LIN {X 0,Y 245.646,Z 172.876,A -85,B 0,C 180,E1 -19098.135,E2 -19098.135} C_VEL
LIN {X 0,Y 243.166,Z 173.176,A -85,B 0,C 180,E1 -19099.924,E2 -19099.924} C_VEL
LIN {X 0,Y 242.08,Z 173.312,A -85,B 0,C 180,E1 -19101.313,E2 -19101.313} C_VEL
LIN {X 0,Y 241.982,Z 173.328,A -85,B 0,C 180,E1 -19101.785,E2 -19101.785} C_VEL
LIN {X 0,Y 241.988,Z 173.343,A -85,B 0,C 180,E1 -19105.826,E2 -19105.826} C_VEL
LIN {X 0,Y 241.964,Z 173.344,A -85,B 0,C 180,E1 -19109.589,E2 -19109.589} C_VEL
LIN {X 0,Y 241.98,Z 173.342,A -85,B 0,C 180,E1 -19113.493,E2 -19113.493} C_VEL
LIN {X 0,Y 241.985,Z 173.344,A -85,B 0,C 180,E1 -19117.583,E2 -19117.583} C_VEL
LIN {X 0,Y 241.909,Z 173.35,A -85,B 0,C 180,E1 -19121.928,E2 -19121.928} C_VEL
LIN {X 0,Y 241.902,Z 173.348,A -85,B 0,C 180,E1 -19126.58,E2 -19126.58} C_VEL
LIN {X 0,Y 241.993,Z 173.342,A -85,B 0,C 180,E1 -19131.641,E2 -19131.641} C_VEL
LIN {X 0,Y 242.055,Z 173.351,A -85,B 0,C 180,E1 -19133.453,E2 -19133.453} C_VEL
LIN {X 0,Y 244.108,Z 182.855,A -85,B 0,C 180,E1 -19137.329,E2 -19137.329} C_VEL
LIN {X 0,Y 244.835,Z 186.515,A -85,B 0,C 180,E1 -19138.763,E2 -19138.763} C_VEL
LIN {X 0,Y 252.464,Z 207.324,A -85,B 0,C 180,E1 -19140.307,E2 -19140.307} C_VEL
LIN {X 0,Y 256.373,Z 235.384,A -85,B 0,C 180,E1 -19141.627,E2 -19141.627} C_VEL
LIN {X 0,Y 254.176,Z 295.63,A -85,B 0,C 180,E1 -19143.433,E2 -19143.433} C_VEL
LIN {X 0,Y 253.102,Z 309.545,A -85,B 0,C 180,E1 -19144.176,E2 -19144.176} C_VEL
LIN {X 0,Y 251.698,Z 321.703,A -85,B 0,C 180,E1 -19145.129,E2 -19145.129} C_VEL
LIN {X 0,Y 250.002,Z 333.498,A -85,B 0,C 180,E1 -19146.385,E2 -19146.385} C_VEL
LIN {X 0,Y 248.104,Z 344.903,A -85,B 0,C 180,E1 -19147.955,E2 -19147.955} C_VEL
LIN {X 0,Y 246.364,Z 355.221,A -85,B 0,C 180,E1 -19149.764,E2 -19149.764} C_VEL
LIN {X 0,Y 244.557,Z 365.313,A -85,B 0,C 180,E1 -19152.005,E2 -19152.005} C_VEL
LIN {X 0,Y 242.888,Z 374.18,A -85,B 0,C 180,E1 -19154.475,E2 -19154.475} C_VEL
LIN {X 0,Y 241.493,Z 381.221,A -85,B 0,C 180,E1 -19156.965,E2 -19156.965} C_VEL
LIN {X 0,Y 240.541,Z 387.674,A -85,B 0,C 180,E1 -19159.904,E2 -19159.904} C_VEL
LIN {X 0,Y 240.047,Z 391.882,A -85,B 0,C 180,E1 -19162.429,E2 -19162.429} C_VEL
LIN {X 0,Y 239.837,Z 395.125,A -85,B 0,C 180,E1 -19165.077,E2 -19165.077} C_VEL
LIN {X 0,Y 239.798,Z 396.531,A -85,B 0,C 180,E1 -19166.64,E2 -19166.64} C_VEL
LIN {X 0,Y 239.844,Z 397.601,A -85,B 0,C 180,E1 -19168.321,E2 -19168.321} C_VEL
LIN {X 0,Y 239.913,Z 398.261,A -85,B 0,C 180,E1 -19170,E2 -19170} C_VEL
LIN {X 0,Y 239.83,Z 398.521,A -85,B 0,C 180,E1 -19171.679,E2 -19171.679} C_VEL
LIN {X 0,Y 239.791,Z 397.941,A -85,B 0,C 180,E1 -19174.792,E2 -19174.792} C_VEL
LIN {X 0,Y 239.953,Z 396.852,A -85,B 0,C 180,E1 -19176.728,E2 -19176.728} C_VEL
LIN {X 0,Y 240.668,Z 393.726,A -85,B 0,C 180,E1 -19180.091,E2 -19180.091} C_VEL
LIN {X 0,Y 241.609,Z 390.211,A -85,B 0,C 180,E1 -19182.601,E2 -19182.601} C_VEL
LIN {X 0,Y 242.969,Z 385.623,A -85,B 0,C 180,E1 -19185.09,E2 -19185.09} C_VEL
LIN {X 0,Y 245.261,Z 378.7,A -85,B 0,C 180,E1 -19187.942,E2 -19187.942} C_VEL
LIN {X 0,Y 247.484,Z 371.049,A -85,B 0,C 180,E1 -19190.425,E2 -19190.425} C_VEL
LIN {X 0,Y 250.137,Z 362.038,A -85,B 0,C 180,E1 -19192.726,E2 -19192.726} C_VEL
LIN {X 0,Y 252.83,Z 352.498,A -85,B 0,C 180,E1 -19194.643,E2 -19194.643} C_VEL
LIN {X 0,Y 255.464,Z 341.974,A -85,B 0,C 180,E1 -19196.335,E2 -19196.335} C_VEL
LIN {X 0,Y 258.126,Z 330.254,A -85,B 0,C 180,E1 -19197.792,E2 -19197.792} C_VEL
LIN {X 0,Y 260.337,Z 317.845,A -85,B 0,C 180,E1 -19198.963,E2 -19198.963} C_VEL
LIN {X 0,Y 262.108,Z 305.644,A -85,B 0,C 180,E1 -19199.795,E2 -19199.795} C_VEL
LIN {X 0,Y 263.402,Z 292.249,A -85,B 0,C 180,E1 -19200.406,E2 -19200.406} C_VEL
LIN {X 0,Y 265.957,Z 237.913,A -85,B 0,C 180,E1 -19202.004,E2 -19202.004} C_VEL
LIN {X 0,Y 263.486,Z 220.784,A -85,B 0,C 180,E1 -19203.076,E2 -19203.076} C_VEL
LIN {X 0,Y 257.206,Z 206.553,A -85,B 0,C 180,E1 -19204.794,E2 -19204.794} C_VEL
LIN {X 0,Y 251.031,Z 194.528,A -85,B 0,C 180,E1 -19206.568,E2 -19206.568} C_VEL
LIN {X 0,Y 247.245,Z 188.246,A -85,B 0,C 180,E1 -19207.687,E2 -19207.687} C_VEL
LIN {X 0,Y 245.239,Z 184.526,A -85,B 0,C 180,E1 -19208.326,E2 -19208.326} C_VEL
LIN {X 0,Y 243.191,Z 177.489,A -85,B 0,C 180,E1 -19212.12,E2 -19212.12} C_VEL
LIN {X 0,Y 241.928,Z 173.348,A -85,B 0,C 180,E1 -19214.685,E2 -19214.685} C_VEL
LIN {X 0,Y 241.914,Z 173.349,A -85,B 0,C 180,E1 -19219.056,E2 -19219.056} C_VEL
LIN {X 0,Y 241.984,Z 173.338,A -85,B 0,C 180,E1 -19222.417,E2 -19222.417} C_VEL
LIN {X 0,Y 241.981,Z 173.333,A -85,B 0,C 180,E1 -19226.507,E2 -19226.507} C_VEL
LIN {X 0,Y 241.972,Z 173.331,A -85,B 0,C 180,E1 -19230.616,E2 -19230.616} C_VEL
LIN {X 0,Y 241.997,Z 173.33,A -85,B 0,C 180,E1 -19234.198,E2 -19234.198} C_VEL
LIN {X 0,Y 241.987,Z 173.333,A -85,B 0,C 180,E1 -19238.338,E2 -19238.338} C_VEL
LIN {X 0,Y 242.108,Z 173.317,A -85,B 0,C 180,E1 -19243.325,E2 -19243.325} C_VEL
LIN {X 0,Y 242.151,Z 173.308,A -85,B 0,C 180,E1 -19248.278,E2 -19248.278} C_VEL
LIN {X 0,Y 242.389,Z 173.289,A -85,B 0,C 180,E1 -19251.664,E2 -19251.664} C_VEL
LIN {X 0,Y 242.408,Z 173.273,A -85,B 0,C 180,E1 -19253.34,E2 -19253.34} C_VEL
LIN {X 0,Y 242.618,Z 173.25,A -85,B 0,C 180,E1 -19258.34,E2 -19258.34} C_VEL
LIN {X 0,Y 242.618,Z 173.251,A -85,B 0,C 180,E1 -19261.66,E2 -19261.66} C_VEL
LIN {X 0,Y 242.403,Z 173.284,A -85,B 0,C 180,E1 -19266.66,E2 -19266.66} C_VEL
LIN {X 0,Y 242.263,Z 173.301,A -85,B 0,C 180,E1 -19270.024,E2 -19270.024} C_VEL
LIN {X 0,Y 242.109,Z 173.323,A -85,B 0,C 180,E1 -19275.145,E2 -19275.145} C_VEL
LIN {X 0,Y 242.076,Z 173.453,A -85,B 0,C 180,E1 -19277.639,E2 -19277.639} C_VEL
LIN {X 0,Y 242.773,Z 175.92,A -85,B 0,C 180,E1 -19279.116,E2 -19279.116} C_VEL
LIN {X 0,Y 245.193,Z 179.843,A -85,B 0,C 180,E1 -19279.9,E2 -19279.9} C_VEL
LIN {X 0,Y 250.376,Z 187.916,A -85,B 0,C 180,E1 -19281.458,E2 -19281.458} C_VEL
LIN {X 0,Y 256.429,Z 198.44,A -85,B 0,C 180,E1 -19283.176,E2 -19283.176} C_VEL
LIN {X 0,Y 262.613,Z 210.801,A -85,B 0,C 180,E1 -19284.837,E2 -19284.837} C_VEL
LIN {X 0,Y 266.786,Z 220.657,A -85,B 0,C 180,E1 -19285.946,E2 -19285.946} C_VEL
LIN {X 0,Y 263.559,Z 283.684,A -85,B 0,C 180,E1 -19287.801,E2 -19287.801} C_VEL
LIN {X 0,Y 262.233,Z 296.967,A -85,B 0,C 180,E1 -19288.483,E2 -19288.483} C_VEL
LIN {X 0,Y 260.633,Z 309.3,A -85,B 0,C 180,E1 -19289.433,E2 -19289.433} C_VEL
LIN {X 0,Y 258.485,Z 321.395,A -85,B 0,C 180,E1 -19290.688,E2 -19290.688} C_VEL
LIN {X 0,Y 256.148,Z 332.007,A -85,B 0,C 180,E1 -19292.098,E2 -19292.098} C_VEL
LIN {X 0,Y 253.657,Z 342.027,A -85,B 0,C 180,E1 -19293.777,E2 -19293.777} C_VEL
LIN {X 0,Y 251.1,Z 351.324,A -85,B 0,C 180,E1 -19295.739,E2 -19295.739} C_VEL
LIN {X 0,Y 248.786,Z 358.929,A -85,B 0,C 180,E1 -19297.722,E2 -19297.722} C_VEL
LIN {X 0,Y 246.429,Z 366.325,A -85,B 0,C 180,E1 -19300.131,E2 -19300.131} C_VEL
LIN {X 0,Y 244.297,Z 372.773,A -85,B 0,C 180,E1 -19302.812,E2 -19302.812} C_VEL
LIN {X 0,Y 242.383,Z 378.302,A -85,B 0,C 180,E1 -19305.901,E2 -19305.901} C_VEL
LIN {X 0,Y 241.425,Z 381.072,A -85,B 0,C 180,E1 -19307.968,E2 -19307.968} C_VEL
LIN {X 0,Y 240.702,Z 383.099,A -85,B 0,C 180,E1 -19310.032,E2 -19310.032} C_VEL
LIN {X 0,Y 240.069,Z 384.596,A -85,B 0,C 180,E1 -19312.225,E2 -19312.225} C_VEL
LIN {X 0,Y 239.587,Z 385.494,A -85,B 0,C 180,E1 -19315.22,E2 -19315.22} C_VEL
LIN {X 0,Y 239.436,Z 385.099,A -85,B 0,C 180,E1 -19318.345,E2 -19318.345} C_VEL
LIN {X 0,Y 239.493,Z 384.301,A -85,B 0,C 180,E1 -19320.074,E2 -19320.074} C_VEL
LIN {X 0,Y 239.701,Z 382.835,A -85,B 0,C 180,E1 -19322.023,E2 -19322.023} C_VEL
LIN {X 0,Y 240.304,Z 379.465,A -85,B 0,C 180,E1 -19325.045,E2 -19325.045} C_VEL
LIN {X 0,Y 240.978,Z 375.219,A -85,B 0,C 180,E1 -19327.719,E2 -19327.719} C_VEL
LIN {X 0,Y 241.958,Z 369.369,A -85,B 0,C 180,E1 -19330.486,E2 -19330.486} C_VEL
LIN {X 0,Y 243.365,Z 361.912,A -85,B 0,C 180,E1 -19333.215,E2 -19333.215} C_VEL
LIN {X 0,Y 244.887,Z 354.288,A -85,B 0,C 180,E1 -19335.433,E2 -19335.433} C_VEL
LIN {X 0,Y 246.618,Z 344.762,A -85,B 0,C 180,E1 -19337.659,E2 -19337.659} C_VEL
LIN {X 0,Y 248.535,Z 334.204,A -85,B 0,C 180,E1 -19339.614,E2 -19339.614} C_VEL
LIN {X 0,Y 250.384,Z 322.487,A -85,B 0,C 180,E1 -19341.324,E2 -19341.324} C_VEL
LIN {X 0,Y 251.952,Z 310.311,A -85,B 0,C 180,E1 -19342.688,E2 -19342.688} C_VEL
LIN {X 0,Y 253.267,Z 297.726,A -85,B 0,C 180,E1 -19343.741,E2 -19343.741} C_VEL
LIN {X 0,Y 254.329,Z 284.519,A -85,B 0,C 180,E1 -19344.485,E2 -19344.485} C_VEL
LIN {X 0,Y 255.167,Z 264.929,A -85,B 0,C 180,E1 -19345.129,E2 -19345.129} C_VEL
LIN {X 0,Y 257.003,Z 212.02,A -85,B 0,C 180,E1 -19346.679,E2 -19346.679} C_VEL
LIN {X 0,Y 251.113,Z 195.487,A -85,B 0,C 180,E1 -19347.835,E2 -19347.835} C_VEL
LIN {X 0,Y 242.82,Z 174.317,A -85,B 0,C 180,E1 -19349.534,E2 -19349.534} C_VEL
LIN {X 0,Y 242.641,Z 173.263,A -85,B 0,C 180,E1 -19350,E2 -19350} C_VEL
LIN {X 0,Y 242.623,Z 173.262,A -85,B 0,C 180,E1 -19351.66,E2 -19351.66} C_VEL
LIN {X 0,Y 242.403,Z 173.288,A -85,B 0,C 180,E1 -19356.66,E2 -19356.66} C_VEL
LIN {X 0,Y 242.268,Z 173.306,A -85,B 0,C 180,E1 -19360.024,E2 -19360.024} C_VEL
LIN {X 0,Y 242.113,Z 173.324,A -85,B 0,C 180,E1 -19365.144,E2 -19365.144} C_VEL
LIN {X 0,Y 242.046,Z 173.333,A -85,B 0,C 180,E1 -19368.626,E2 -19368.626} C_VEL
LIN {X 0,Y 241.99,Z 173.337,A -85,B 0,C 180,E1 -19372.182,E2 -19372.182} C_VEL
LIN {X 0,Y 241.988,Z 173.336,A -85,B 0,C 180,E1 -19375.826,E2 -19375.826} C_VEL
LIN {X 0,Y 241.97,Z 173.344,A -85,B 0,C 180,E1 -19379.588,E2 -19379.588} C_VEL
LIN {X 0,Y 241.981,Z 173.326,A -85,B 0,C 180,E1 -19383.493,E2 -19383.493} C_VEL
LIN {X 0,Y 241.988,Z 173.341,A -85,B 0,C 180,E1 -19387.583,E2 -19387.583} C_VEL
LIN {X 0,Y 241.911,Z 173.346,A -85,B 0,C 180,E1 -19391.928,E2 -19391.928} C_VEL
LIN {X 0,Y 241.902,Z 173.325,A -85,B 0,C 180,E1 -19396.58,E2 -19396.58} C_VEL
LIN {X 0,Y 241.995,Z 173.339,A -85,B 0,C 180,E1 -19401.641,E2 -19401.641} C_VEL
LIN {X 0,Y 241.982,Z 173.342,A -85,B 0,C 180,E1 -19404.488,E2 -19404.488} C_VEL
LIN {X 0,Y 241.955,Z 173.337,A -85,B 0,C 180,E1 -19408.477,E2 -19408.477} C_VEL
LIN {X 0,Y 241.97,Z 173.343,A -85,B 0,C 180,E1 -19412.308,E2 -19412.308} C_VEL
LIN {X 0,Y 242.026,Z 173.33,A -85,B 0,C 180,E1 -19416.012,E2 -19416.012} C_VEL
LIN {X 0,Y 241.987,Z 173.339,A -85,B 0,C 180,E1 -19419.603,E2 -19419.603} C_VEL
LIN {X 0,Y 242.108,Z 173.322,A -85,B 0,C 180,E1 -19423.324,E2 -19423.324} C_VEL
LIN {X 0,Y 242.164,Z 173.318,A -85,B 0,C 180,E1 -19428.279,E2 -19428.279} C_VEL
LIN {X 0,Y 242.388,Z 173.289,A -85,B 0,C 180,E1 -19431.664,E2 -19431.664} C_VEL
LIN {X 0,Y 242.404,Z 173.283,A -85,B 0,C 180,E1 -19433.34,E2 -19433.34} C_VEL
LIN {X 0,Y 242.62,Z 173.265,A -85,B 0,C 180,E1 -19438.34,E2 -19438.34} C_VEL
LIN {X 0,Y 242.619,Z 173.259,A -85,B 0,C 180,E1 -19441.66,E2 -19441.66} C_VEL
LIN {X 0,Y 242.399,Z 173.263,A -85,B 0,C 180,E1 -19446.66,E2 -19446.66} C_VEL
LIN {X 0,Y 242.262,Z 173.298,A -85,B 0,C 180,E1 -19450.024,E2 -19450.024} C_VEL
LIN {X 0,Y 242.104,Z 173.326,A -85,B 0,C 180,E1 -19455.145,E2 -19455.145} C_VEL
LIN {X 0,Y 242.016,Z 173.325,A -85,B 0,C 180,E1 -19458.629,E2 -19458.629} C_VEL
LIN {X 0,Y 241.982,Z 173.328,A -85,B 0,C 180,E1 -19461.785,E2 -19461.785} C_VEL
LIN {X 0,Y 241.28,Z 173.426,A -85,B 0,C 180,E1 -19463.175,E2 -19463.175} C_VEL
LIN {X 0,Y 238.396,Z 173.79,A -85,B 0,C 180,E1 -19465.442,E2 -19465.442} C_VEL
LIN {X 0,Y 235.978,Z 174.091,A -85,B 0,C 180,E1 -19467.289,E2 -19467.289} C_VEL
LIN {X 0,Y 234.964,Z 174.212,A -85,B 0,C 180,E1 -19468.723,E2 -19468.723} C_VEL
LIN {X 0,Y 234.893,Z 174.221,A -85,B 0,C 180,E1 -19469.208,E2 -19469.208} C_VEL
LIN {X 0,Y 234.942,Z 174.22,A -85,B 0,C 180,E1 -19473.113,E2 -19473.113} C_VEL
LIN {X 0,Y 234.917,Z 174.224,A -85,B 0,C 180,E1 -19476.751,E2 -19476.751} C_VEL
LIN {X 0,Y 234.913,Z 174.225,A -85,B 0,C 180,E1 -19478.935,E2 -19478.935} C_VEL
LIN {X 0,Y 234.854,Z 174.23,A -85,B 0,C 180,E1 -19483.494,E2 -19483.494} C_VEL
LIN {X 0,Y 234.855,Z 174.226,A -85,B 0,C 180,E1 -19486.506,E2 -19486.506} C_VEL
LIN {X 0,Y 234.919,Z 174.224,A -85,B 0,C 180,E1 -19491.078,E2 -19491.078} C_VEL
LIN {X 0,Y 234.993,Z 174.243,A -85,B 0,C 180,E1 -19492.861,E2 -19492.861} C_VEL
LIN {X 0,Y 237.063,Z 183.657,A -85,B 0,C 180,E1 -19496.833,E2 -19496.833} C_VEL
LIN {X 0,Y 237.643,Z 186.548,A -85,B 0,C 180,E1 -19497.927,E2 -19497.927} C_VEL
LIN {X 0,Y 246.115,Z 209.016,A -85,B 0,C 180,E1 -19499.693,E2 -19499.693} C_VEL
LIN {X 0,Y 249.791,Z 235.832,A -85,B 0,C 180,E1 -19500.997,E2 -19500.997} C_VEL
LIN {X 0,Y 247.639,Z 294.718,A -85,B 0,C 180,E1 -19502.803,E2 -19502.803} C_VEL
LIN {X 0,Y 246.541,Z 308.656,A -85,B 0,C 180,E1 -19503.55,E2 -19503.55} C_VEL
LIN {X 0,Y 245.09,Z 321.021,A -85,B 0,C 180,E1 -19504.524,E2 -19504.524} C_VEL
LIN {X 0,Y 243.504,Z 332.149,A -85,B 0,C 180,E1 -19505.714,E2 -19505.714} C_VEL
LIN {X 0,Y 241.543,Z 343.765,A -85,B 0,C 180,E1 -19507.323,E2 -19507.323} C_VEL
LIN {X 0,Y 239.639,Z 354.257,A -85,B 0,C 180,E1 -19509.17,E2 -19509.17} C_VEL
LIN {X 0,Y 237.983,Z 362.832,A -85,B 0,C 180,E1 -19511.044,E2 -19511.044} C_VEL
LIN {X 0,Y 236.495,Z 370.734,A -85,B 0,C 180,E1 -19513.157,E2 -19513.157} C_VEL
LIN {X 0,Y 234.982,Z 378.423,A -85,B 0,C 180,E1 -19515.715,E2 -19515.715} C_VEL
LIN {X 0,Y 233.779,Z 385.517,A -85,B 0,C 180,E1 -19518.731,E2 -19518.731} C_VEL
LIN {X 0,Y 233.168,Z 390.19,A -85,B 0,C 180,E1 -19521.332,E2 -19521.332} C_VEL
LIN {X 0,Y 232.896,Z 392.644,A -85,B 0,C 180,E1 -19523.067,E2 -19523.067} C_VEL
LIN {X 0,Y 232.728,Z 395.091,A -85,B 0,C 180,E1 -19525.238,E2 -19525.238} C_VEL
LIN {X 0,Y 232.756,Z 397.333,A -85,B 0,C 180,E1 -19528.27,E2 -19528.27} C_VEL
LIN {X 0,Y 232.823,Z 398.022,A -85,B 0,C 180,E1 -19530,E2 -19530} C_VEL
LIN {X 0,Y 232.742,Z 398.31,A -85,B 0,C 180,E1 -19531.73,E2 -19531.73} C_VEL
LIN {X 0,Y 232.707,Z 397.869,A -85,B 0,C 180,E1 -19534.699,E2 -19534.699} C_VEL
LIN {X 0,Y 232.891,Z 396.752,A -85,B 0,C 180,E1 -19536.933,E2 -19536.933} C_VEL
LIN {X 0,Y 233.665,Z 393.688,A -85,B 0,C 180,E1 -19540.397,E2 -19540.397} C_VEL
LIN {X 0,Y 234.644,Z 390.234,A -85,B 0,C 180,E1 -19542.982,E2 -19542.982} C_VEL
LIN {X 0,Y 236.127,Z 385.723,A -85,B 0,C 180,E1 -19545.538,E2 -19545.538} C_VEL
LIN {X 0,Y 238.511,Z 378.933,A -85,B 0,C 180,E1 -19548.467,E2 -19548.467} C_VEL
LIN {X 0,Y 240.749,Z 371.719,A -85,B 0,C 180,E1 -19550.908,E2 -19550.908} C_VEL
LIN {X 0,Y 243.622,Z 362.498,A -85,B 0,C 180,E1 -19553.37,E2 -19553.37} C_VEL
LIN {X 0,Y 246.725,Z 352.045,A -85,B 0,C 180,E1 -19555.521,E2 -19555.521} C_VEL
LIN {X 0,Y 249.52,Z 341.464,A -85,B 0,C 180,E1 -19557.239,E2 -19557.239} C_VEL
LIN {X 0,Y 252.245,Z 329.657,A -85,B 0,C 180,E1 -19558.726,E2 -19558.726} C_VEL
LIN {X 0,Y 254.564,Z 317.191,A -85,B 0,C 180,E1 -19559.912,E2 -19559.912} C_VEL
LIN {X 0,Y 256.523,Z 304.129,A -85,B 0,C 180,E1 -19560.796,E2 -19560.796} C_VEL
LIN {X 0,Y 257.782,Z 290.61,A -85,B 0,C 180,E1 -19561.392,E2 -19561.392} C_VEL
LIN {X 0,Y 260.312,Z 238.633,A -85,B 0,C 180,E1 -19562.955,E2 -19562.955} C_VEL
LIN {X 0,Y 258.26,Z 223.958,A -85,B 0,C 180,E1 -19563.902,E2 -19563.902} C_VEL
LIN {X 0,Y 252.636,Z 210.85,A -85,B 0,C 180,E1 -19565.538,E2 -19565.538} C_VEL
LIN {X 0,Y 246.677,Z 199.127,A -85,B 0,C 180,E1 -19567.332,E2 -19567.332} C_VEL
LIN {X 0,Y 240.762,Z 188.999,A -85,B 0,C 180,E1 -19569.226,E2 -19569.226} C_VEL
LIN {X 0,Y 238.016,Z 184.471,A -85,B 0,C 180,E1 -19570.159,E2 -19570.159} C_VEL
LIN {X 0,Y 236.345,Z 179.132,A -85,B 0,C 180,E1 -19573.152,E2 -19573.152} C_VEL
LIN {X 0,Y 234.862,Z 174.229,A -85,B 0,C 180,E1 -19576.277,E2 -19576.277} C_VEL
LIN {X 0,Y 234.919,Z 174.219,A -85,B 0,C 180,E1 -19581.079,E2 -19581.079} C_VEL
LIN {X 0,Y 234.927,Z 174.221,A -85,B 0,C 180,E1 -19585.361,E2 -19585.361} C_VEL
LIN {X 0,Y 234.897,Z 174.222,A -85,B 0,C 180,E1 -19589.427,E2 -19589.427} C_VEL
LIN {X 0,Y 234.941,Z 174.213,A -85,B 0,C 180,E1 -19593.822,E2 -19593.822} C_VEL
LIN {X 0,Y 234.937,Z 174.206,A -85,B 0,C 180,E1 -19598.963,E2 -19598.963} C_VEL
LIN {X 0,Y 235.052,Z 174.197,A -85,B 0,C 180,E1 -19603.098,E2 -19603.098} C_VEL
LIN {X 0,Y 235.083,Z 174.191,A -85,B 0,C 180,E1 -19607.92,E2 -19607.92} C_VEL
LIN {X 0,Y 235.319,Z 174.17,A -85,B 0,C 180,E1 -19611.412,E2 -19611.412} C_VEL
LIN {X 0,Y 235.36,Z 174.151,A -85,B 0,C 180,E1 -19613.14,E2 -19613.14} C_VEL
LIN {X 0,Y 235.577,Z 174.126,A -85,B 0,C 180,E1 -19618.291,E2 -19618.291} C_VEL
LIN {X 0,Y 235.577,Z 174.128,A -85,B 0,C 180,E1 -19621.71,E2 -19621.71} C_VEL
LIN {X 0,Y 235.355,Z 174.163,A -85,B 0,C 180,E1 -19626.86,E2 -19626.86} C_VEL
LIN {X 0,Y 235.187,Z 174.185,A -85,B 0,C 180,E1 -19630.329,E2 -19630.329} C_VEL
LIN {X 0,Y 235.045,Z 174.202,A -85,B 0,C 180,E1 -19635.611,E2 -19635.611} C_VEL
LIN {X 0,Y 235.091,Z 174.366,A -85,B 0,C 180,E1 -19636.002,E2 -19636.002} C_VEL
LIN {X 0,Y 235.709,Z 176.425,A -85,B 0,C 180,E1 -19637.256,E2 -19637.256} C_VEL
LIN {X 0,Y 238.369,Z 180.619,A -85,B 0,C 180,E1 -19638.201,E2 -19638.201} C_VEL
LIN {X 0,Y 242.949,Z 187.493,A -85,B 0,C 180,E1 -19639.706,E2 -19639.706} C_VEL
LIN {X 0,Y 248.169,Z 196.06,A -85,B 0,C 180,E1 -19641.323,E2 -19641.323} C_VEL
LIN {X 0,Y 253.917,Z 206.683,A -85,B 0,C 180,E1 -19643.005,E2 -19643.005} C_VEL
LIN {X 0,Y 259.476,Z 218.638,A -85,B 0,C 180,E1 -19644.568,E2 -19644.568} C_VEL
LIN {X 0,Y 261.085,Z 222.691,A -85,B 0,C 180,E1 -19645.02,E2 -19645.02} C_VEL
LIN {X 0,Y 257.905,Z 283.565,A -85,B 0,C 180,E1 -19646.857,E2 -19646.857} C_VEL
LIN {X 0,Y 256.434,Z 297.541,A -85,B 0,C 180,E1 -19647.586,E2 -19647.586} C_VEL
LIN {X 0,Y 254.666,Z 310.279,A -85,B 0,C 180,E1 -19648.606,E2 -19648.606} C_VEL
LIN {X 0,Y 252.325,Z 322.628,A -85,B 0,C 180,E1 -19649.937,E2 -19649.937} C_VEL
LIN {X 0,Y 249.563,Z 334.369,A -85,B 0,C 180,E1 -19651.583,E2 -19651.583} C_VEL
LIN {X 0,Y 246.641,Z 345.145,A -85,B 0,C 180,E1 -19653.542,E2 -19653.542} C_VEL
LIN {X 0,Y 244.028,Z 353.961,A -85,B 0,C 180,E1 -19655.565,E2 -19655.565} C_VEL
LIN {X 0,Y 241.148,Z 362.711,A -85,B 0,C 180,E1 -19658.104,E2 -19658.104} C_VEL
LIN {X 0,Y 238.708,Z 369.857,A -85,B 0,C 180,E1 -19660.783,E2 -19660.783} C_VEL
LIN {X 0,Y 236.544,Z 375.828,A -85,B 0,C 180,E1 -19663.699,E2 -19663.699} C_VEL
LIN {X 0,Y 234.947,Z 380.079,A -85,B 0,C 180,E1 -19666.527,E2 -19666.527} C_VEL
LIN {X 0,Y 234.046,Z 382.445,A -85,B 0,C 180,E1 -19668.652,E2 -19668.652} C_VEL
LIN {X 0,Y 233.109,Z 384.665,A -85,B 0,C 180,E1 -19671.617,E2 -19671.617} C_VEL
LIN {X 0,Y 232.511,Z 385.692,A -85,B 0,C 180,E1 -19674.949,E2 -19674.949} C_VEL
LIN {X 0,Y 232.331,Z 385.392,A -85,B 0,C 180,E1 -19677.887,E2 -19677.887} C_VEL
LIN {X 0,Y 232.505,Z 383.664,A -85,B 0,C 180,E1 -19681.235,E2 -19681.235} C_VEL
LIN {X 0,Y 232.792,Z 382.025,A -85,B 0,C 180,E1 -19683.073,E2 -19683.073} C_VEL
LIN {X 0,Y 233.426,Z 378.376,A -85,B 0,C 180,E1 -19686.017,E2 -19686.017} C_VEL
LIN {X 0,Y 234.209,Z 373.461,A -85,B 0,C 180,E1 -19688.894,E2 -19688.894} C_VEL
LIN {X 0,Y 235.403,Z 367.094,A -85,B 0,C 180,E1 -19691.723,E2 -19691.723} C_VEL
LIN {X 0,Y 237.087,Z 358.903,A -85,B 0,C 180,E1 -19694.527,E2 -19694.527} C_VEL
LIN {X 0,Y 238.796,Z 350.205,A -85,B 0,C 180,E1 -19696.89,E2 -19696.89} C_VEL
LIN {X 0,Y 240.711,Z 340.105,A -85,B 0,C 180,E1 -19699.06,E2 -19699.06} C_VEL
LIN {X 0,Y 242.722,Z 328.611,A -85,B 0,C 180,E1 -19701.014,E2 -19701.014} C_VEL
LIN {X 0,Y 244.479,Z 316.777,A -85,B 0,C 180,E1 -19702.567,E2 -19702.567} C_VEL
LIN {X 0,Y 245.903,Z 304.915,A -85,B 0,C 180,E1 -19703.763,E2 -19703.763} C_VEL
LIN {X 0,Y 247.216,Z 292.061,A -85,B 0,C 180,E1 -19704.698,E2 -19704.698} C_VEL
LIN {X 0,Y 248.07,Z 279.034,A -85,B 0,C 180,E1 -19705.31,E2 -19705.31} C_VEL
LIN {X 0,Y 250.551,Z 213.75,A -85,B 0,C 180,E1 -19707.274,E2 -19707.274} C_VEL
LIN {X 0,Y 244.449,Z 196.814,A -85,B 0,C 180,E1 -19708.517,E2 -19708.517} C_VEL
LIN {X 0,Y 236.783,Z 177.405,A -85,B 0,C 180,E1 -19710.106,E2 -19710.106} C_VEL
LIN {X 0,Y 235.623,Z 174.45,A -85,B 0,C 180,E1 -19710.427,E2 -19710.427} C_VEL
LIN {X 0,Y 235.563,Z 174.14,A -85,B 0,C 180,E1 -19710.855,E2 -19710.855} C_VEL
LIN {X 0,Y 235.191,Z 174.191,A -85,B 0,C 180,E1 -19715.143,E2 -19715.143} C_VEL
LIN {X 0,Y 235.356,Z 174.166,A -85,B 0,C 180,E1 -19716.86,E2 -19716.86} C_VEL
LIN {X 0,Y 235.213,Z 174.182,A -85,B 0,C 180,E1 -19720.328,E2 -19720.328} C_VEL
LIN {X 0,Y 235.065,Z 174.2,A -85,B 0,C 180,E1 -19725.61,E2 -19725.61} C_VEL
LIN {X 0,Y 234.987,Z 174.213,A -85,B 0,C 180,E1 -19729.208,E2 -19729.208} C_VEL
LIN {X 0,Y 234.918,Z 174.216,A -85,B 0,C 180,E1 -19732.887,E2 -19732.887} C_VEL
LIN {X 0,Y 234.928,Z 174.218,A -85,B 0,C 180,E1 -19736.663,E2 -19736.663} C_VEL
LIN {X 0,Y 234.9,Z 174.22,A -85,B 0,C 180,E1 -19740.572,E2 -19740.572} C_VEL
LIN {X 0,Y 234.931,Z 174.205,A -85,B 0,C 180,E1 -19744.638,E2 -19744.638} C_VEL
LIN {X 0,Y 234.913,Z 174.222,A -85,B 0,C 180,E1 -19748.935,E2 -19748.935} C_VEL
LIN {X 0,Y 234.855,Z 174.218,A -85,B 0,C 180,E1 -19753.494,E2 -19753.494} C_VEL
LIN {X 0,Y 234.854,Z 174.201,A -85,B 0,C 180,E1 -19756.506,E2 -19756.506} C_VEL
LIN {X 0,Y 234.919,Z 174.217,A -85,B 0,C 180,E1 -19761.079,E2 -19761.079} C_VEL
LIN {X 0,Y 234.928,Z 174.219,A -85,B 0,C 180,E1 -19765.361,E2 -19765.361} C_VEL
LIN {X 0,Y 234.901,Z 174.221,A -85,B 0,C 180,E1 -19769.428,E2 -19769.428} C_VEL
LIN {X 0,Y 234.971,Z 174.213,A -85,B 0,C 180,E1 -19773.807,E2 -19773.807} C_VEL
LIN {X 0,Y 234.967,Z 174.21,A -85,B 0,C 180,E1 -19778.008,E2 -19778.008} C_VEL
LIN {X 0,Y 235.052,Z 174.202,A -85,B 0,C 180,E1 -19783.098,E2 -19783.098} C_VEL
LIN {X 0,Y 235.094,Z 174.197,A -85,B 0,C 180,E1 -19787.921,E2 -19787.921} C_VEL
LIN {X 0,Y 235.322,Z 174.169,A -85,B 0,C 180,E1 -19791.412,E2 -19791.412} C_VEL
LIN {X 0,Y 235.356,Z 174.16,A -85,B 0,C 180,E1 -19793.14,E2 -19793.14} C_VEL
LIN {X 0,Y 235.579,Z 174.142,A -85,B 0,C 180,E1 -19798.29,E2 -19798.29} C_VEL
LIN {X 0,Y 235.578,Z 174.136,A -85,B 0,C 180,E1 -19801.709,E2 -19801.709} C_VEL
LIN {X 0,Y 235.35,Z 174.139,A -85,B 0,C 180,E1 -19806.86,E2 -19806.86} C_VEL
LIN {X 0,Y 235.185,Z 174.182,A -85,B 0,C 180,E1 -19810.329,E2 -19810.329} C_VEL
LIN {X 0,Y 235.057,Z 174.205,A -85,B 0,C 180,E1 -19815.61,E2 -19815.61} C_VEL
LIN {X 0,Y 234.958,Z 174.201,A -85,B 0,C 180,E1 -19819.21,E2 -19819.21} C_VEL
LIN {X 0,Y 234.918,Z 174.213,A -85,B 0,C 180,E1 -19822.887,E2 -19822.887} C_VEL
LIN {X 0,Y 234.924,Z 174.22,A -85,B 0,C 180,E1 -19826.663,E2 -19826.663} C_VEL
LIN {X 0,Y 234.893,Z 174.221,A -85,B 0,C 180,E1 -19829.208,E2 -19829.208} C_VEL
LIN {X 0,Y 234.27,Z 174.306,A -85,B 0,C 180,E1 -19830.639,E2 -19830.639} C_VEL
LIN {X 0,Y 231.481,Z 174.66,A -85,B 0,C 180,E1 -19832.975,E2 -19832.975} C_VEL
LIN {X 0,Y 228.229,Z 175.061,A -85,B 0,C 180,E1 -19835.858,E2 -19835.858} C_VEL
LIN {X 0,Y 227.869,Z 175.101,A -85,B 0,C 180,E1 -19836.857,E2 -19836.857} C_VEL
LIN {X 0,Y 227.802,Z 175.108,A -85,B 0,C 180,E1 -19840.382,E2 -19840.382} C_VEL
LIN {X 0,Y 227.811,Z 175.1,A -85,B 0,C 180,E1 -19845.199,E2 -19845.199} C_VEL
LIN {X 0,Y 227.801,Z 175.103,A -85,B 0,C 180,E1 -19849.618,E2 -19849.618} C_VEL
LIN {X 0,Y 227.943,Z 175.254,A -85,B 0,C 180,E1 -19852.284,E2 -19852.284} C_VEL
LIN {X 0,Y 230.181,Z 185.282,A -85,B 0,C 180,E1 -19856.661,E2 -19856.661} C_VEL
LIN {X 0,Y 230.342,Z 186.077,A -85,B 0,C 180,E1 -19856.995,E2 -19856.995} C_VEL
LIN {X 0,Y 238.882,Z 208.491,A -85,B 0,C 180,E1 -19858.865,E2 -19858.865} C_VEL
LIN {X 0,Y 240.005,Z 212.386,A -85,B 0,C 180,E1 -19859.132,E2 -19859.132} C_VEL
LIN {X 0,Y 243.342,Z 237.389,A -85,B 0,C 180,E1 -19860.382,E2 -19860.382} C_VEL
LIN {X 0,Y 241.058,Z 294.986,A -85,B 0,C 180,E1 -19862.194,E2 -19862.194} C_VEL
LIN {X 0,Y 239.945,Z 308.516,A -85,B 0,C 180,E1 -19862.941,E2 -19862.941} C_VEL
LIN {X 0,Y 238.535,Z 320.317,A -85,B 0,C 180,E1 -19863.889,E2 -19863.889} C_VEL
LIN {X 0,Y 236.741,Z 332.379,A -85,B 0,C 180,E1 -19865.208,E2 -19865.208} C_VEL
LIN {X 0,Y 234.721,Z 343.92,A -85,B 0,C 180,E1 -19866.859,E2 -19866.859} C_VEL
LIN {X 0,Y 232.772,Z 354.354,A -85,B 0,C 180,E1 -19868.758,E2 -19868.758} C_VEL
LIN {X 0,Y 230.806,Z 364.407,A -85,B 0,C 180,E1 -19871.086,E2 -19871.086} C_VEL
LIN {X 0,Y 229.11,Z 372.796,A -85,B 0,C 180,E1 -19873.516,E2 -19873.516} C_VEL
LIN {X 0,Y 227.593,Z 380.08,A -85,B 0,C 180,E1 -19876.154,E2 -19876.154} C_VEL
LIN {X 0,Y 226.762,Z 384.989,A -85,B 0,C 180,E1 -19878.378,E2 -19878.378} C_VEL
LIN {X 0,Y 226.118,Z 389.738,A -85,B 0,C 180,E1 -19881.06,E2 -19881.06} C_VEL
LIN {X 0,Y 225.726,Z 393.332,A -85,B 0,C 180,E1 -19883.744,E2 -19883.744} C_VEL
LIN {X 0,Y 225.618,Z 395.883,A -85,B 0,C 180,E1 -19886.428,E2 -19886.428} C_VEL
LIN {X 0,Y 225.67,Z 397.062,A -85,B 0,C 180,E1 -19888.215,E2 -19888.215} C_VEL
LIN {X 0,Y 225.734,Z 397.783,A -85,B 0,C 180,E1 -19890,E2 -19890} C_VEL
LIN {X 0,Y 225.655,Z 398.099,A -85,B 0,C 180,E1 -19891.785,E2 -19891.785} C_VEL
LIN {X 0,Y 225.647,Z 397.557,A -85,B 0,C 180,E1 -19895.362,E2 -19895.362} C_VEL
LIN {X 0,Y 226.153,Z 395.36,A -85,B 0,C 180,E1 -19898.939,E2 -19898.939} C_VEL
LIN {X 0,Y 226.959,Z 392.642,A -85,B 0,C 180,E1 -19901.612,E2 -19901.612} C_VEL
LIN {X 0,Y 228.122,Z 388.922,A -85,B 0,C 180,E1 -19904.269,E2 -19904.269} C_VEL
LIN {X 0,Y 229.943,Z 384.102,A -85,B 0,C 180,E1 -19906.88,E2 -19906.88} C_VEL
LIN {X 0,Y 232.123,Z 378.045,A -85,B 0,C 180,E1 -19909.454,E2 -19909.454} C_VEL
LIN {X 0,Y 234.633,Z 370.547,A -85,B 0,C 180,E1 -19911.987,E2 -19911.987} C_VEL
LIN {X 0,Y 237.147,Z 362.938,A -85,B 0,C 180,E1 -19914.048,E2 -19914.048} C_VEL
LIN {X 0,Y 240.073,Z 353.766,A -85,B 0,C 180,E1 -19916.048,E2 -19916.048} C_VEL
LIN {X 0,Y 242.92,Z 343.626,A -85,B 0,C 180,E1 -19917.809,E2 -19917.809} C_VEL
LIN {X 0,Y 245.771,Z 332.443,A -85,B 0,C 180,E1 -19919.321,E2 -19919.321} C_VEL
LIN {X 0,Y 248.32,Z 319.976,A -85,B 0,C 180,E1 -19920.627,E2 -19920.627} C_VEL
LIN {X 0,Y 250.32,Z 307.949,A -85,B 0,C 180,E1 -19921.528,E2 -19921.528} C_VEL
LIN {X 0,Y 251.918,Z 294.009,A -85,B 0,C 180,E1 -19922.245,E2 -19922.245} C_VEL
LIN {X 0,Y 254.832,Z 240.209,A -85,B 0,C 180,E1 -19923.898,E2 -19923.898} C_VEL
LIN {X 0,Y 252.983,Z 226.709,A -85,B 0,C 180,E1 -19924.805,E2 -19924.805} C_VEL
LIN {X 0,Y 247.947,Z 214.829,A -85,B 0,C 180,E1 -19926.364,E2 -19926.364} C_VEL
LIN {X 0,Y 242.519,Z 203.911,A -85,B 0,C 180,E1 -19928.088,E2 -19928.088} C_VEL
LIN {X 0,Y 236.701,Z 193.829,A -85,B 0,C 180,E1 -19930.049,E2 -19930.049} C_VEL
LIN {X 0,Y 233.384,Z 188.536,A -85,B 0,C 180,E1 -19931.236,E2 -19931.236} C_VEL
LIN {X 0,Y 230.616,Z 184.055,A -85,B 0,C 180,E1 -19932.29,E2 -19932.29} C_VEL
LIN {X 0,Y 228.661,Z 177.809,A -85,B 0,C 180,E1 -19936.247,E2 -19936.247} C_VEL
LIN {X 0,Y 227.813,Z 175.108,A -85,B 0,C 180,E1 -19938.198,E2 -19938.198} C_VEL
LIN {X 0,Y 227.841,Z 175.104,A -85,B 0,C 180,E1 -19941.908,E2 -19941.908} C_VEL
LIN {X 0,Y 227.88,Z 175.09,A -85,B 0,C 180,E1 -19946.378,E2 -19946.378} C_VEL
LIN {X 0,Y 227.873,Z 175.088,A -85,B 0,C 180,E1 -19950.431,E2 -19950.431} C_VEL
LIN {X 0,Y 227.867,Z 175.088,A -85,B 0,C 180,E1 -19954.418,E2 -19954.418} C_VEL
LIN {X 0,Y 227.921,Z 175.085,A -85,B 0,C 180,E1 -19958.283,E2 -19958.283} C_VEL
LIN {X 0,Y 228.001,Z 175.07,A -85,B 0,C 180,E1 -19963.894,E2 -19963.894} C_VEL
LIN {X 0,Y 228.126,Z 175.052,A -85,B 0,C 180,E1 -19969.348,E2 -19969.348} C_VEL
LIN {X 0,Y 228.311,Z 175.029,A -85,B 0,C 180,E1 -19972.927,E2 -19972.927} C_VEL
LIN {X 0,Y 228.535,Z 175.003,A -85,B 0,C 180,E1 -19978.238,E2 -19978.238} C_VEL
LIN {X 0,Y 228.535,Z 175.005,A -85,B 0,C 180,E1 -19981.762,E2 -19981.762} C_VEL
LIN {X 0,Y 228.307,Z 175.042,A -85,B 0,C 180,E1 -19987.073,E2 -19987.073} C_VEL
LIN {X 0,Y 228.128,Z 175.067,A -85,B 0,C 180,E1 -19990.652,E2 -19990.652} C_VEL
LIN {X 0,Y 228.016,Z 175.171,A -85,B 0,C 180,E1 -19994.048,E2 -19994.048} C_VEL
LIN {X 0,Y 228.476,Z 176.87,A -85,B 0,C 180,E1 -19995.1,E2 -19995.1} C_VEL
LIN {X 0,Y 231.301,Z 180.949,A -85,B 0,C 180,E1 -19996.204,E2 -19996.204} C_VEL
LIN {X 0,Y 232.725,Z 182.905,A -85,B 0,C 180,E1 -19996.734,E2 -19996.734} C_VEL
LIN {X 0,Y 238.966,Z 192.402,A -85,B 0,C 180,E1 -19998.931,E2 -19998.931} C_VEL
LIN {X 0,Y 243.942,Z 200.772,A -85,B 0,C 180,E1 -20000.563,E2 -20000.563} C_VEL
LIN {X 0,Y 249.288,Z 210.737,A -85,B 0,C 180,E1 -20002.205,E2 -20002.205} C_VEL
LIN {X 0,Y 254.724,Z 222.814,A -85,B 0,C 180,E1 -20003.836,E2 -20003.836} C_VEL
LIN {X 0,Y 255.6,Z 224.985,A -85,B 0,C 180,E1 -20004.094,E2 -20004.094} C_VEL
LIN {X 0,Y 252.309,Z 283.774,A -85,B 0,C 180,E1 -20005.883,E2 -20005.883} C_VEL
LIN {X 0,Y 250.848,Z 297.348,A -85,B 0,C 180,E1 -20006.601,E2 -20006.601} C_VEL
LIN {X 0,Y 249.144,Z 309.109,A -85,B 0,C 180,E1 -20007.524,E2 -20007.524} C_VEL
LIN {X 0,Y 246.898,Z 320.904,A -85,B 0,C 180,E1 -20008.769,E2 -20008.769} C_VEL
LIN {X 0,Y 244.209,Z 332.16,A -85,B 0,C 180,E1 -20010.303,E2 -20010.303} C_VEL
LIN {X 0,Y 241.412,Z 342.444,A -85,B 0,C 180,E1 -20012.093,E2 -20012.093} C_VEL
LIN {X 0,Y 238.659,Z 351.307,A -85,B 0,C 180,E1 -20014.022,E2 -20014.022} C_VEL
LIN {X 0,Y 235.472,Z 360.751,A -85,B 0,C 180,E1 -20016.651,E2 -20016.651} C_VEL
LIN {X 0,Y 232.755,Z 368.323,A -85,B 0,C 180,E1 -20019.353,E2 -20019.353} C_VEL
LIN {X 0,Y 230.455,Z 374.305,A -85,B 0,C 180,E1 -20022.138,E2 -20022.138} C_VEL
LIN {X 0,Y 228.629,Z 378.967,A -85,B 0,C 180,E1 -20025.007,E2 -20025.007} C_VEL
LIN {X 0,Y 227.238,Z 382.39,A -85,B 0,C 180,E1 -20027.925,E2 -20027.925} C_VEL
LIN {X 0,Y 226.211,Z 384.697,A -85,B 0,C 180,E1 -20030.961,E2 -20030.961} C_VEL
LIN {X 0,Y 225.522,Z 385.845,A -85,B 0,C 180,E1 -20034.12,E2 -20034.12} C_VEL
LIN {X 0,Y 225.26,Z 385.685,A -85,B 0,C 180,E1 -20037.394,E2 -20037.394} C_VEL
LIN {X 0,Y 225.36,Z 384.087,A -85,B 0,C 180,E1 -20040.833,E2 -20040.833} C_VEL
LIN {X 0,Y 225.9,Z 381.065,A -85,B 0,C 180,E1 -20044.179,E2 -20044.179} C_VEL
LIN {X 0,Y 226.615,Z 376.945,A -85,B 0,C 180,E1 -20047.191,E2 -20047.191} C_VEL
LIN {X 0,Y 227.559,Z 371.507,A -85,B 0,C 180,E1 -20050.14,E2 -20050.14} C_VEL
LIN {X 0,Y 228.968,Z 364.542,A -85,B 0,C 180,E1 -20053.046,E2 -20053.046} C_VEL
LIN {X 0,Y 230.504,Z 357.283,A -85,B 0,C 180,E1 -20055.431,E2 -20055.431} C_VEL
LIN {X 0,Y 232.323,Z 348.425,A -85,B 0,C 180,E1 -20057.775,E2 -20057.775} C_VEL
LIN {X 0,Y 234.272,Z 338.336,A -85,B 0,C 180,E1 -20059.917,E2 -20059.917} C_VEL
LIN {X 0,Y 236.113,Z 328.032,A -85,B 0,C 180,E1 -20061.656,E2 -20061.656} C_VEL
LIN {X 0,Y 237.897,Z 316.281,A -85,B 0,C 180,E1 -20063.213,E2 -20063.213} C_VEL
LIN {X 0,Y 239.417,Z 304.06,A -85,B 0,C 180,E1 -20064.452,E2 -20064.452} C_VEL
LIN {X 0,Y 240.669,Z 291.78,A -85,B 0,C 180,E1 -20065.344,E2 -20065.344} C_VEL
LIN {X 0,Y 241.527,Z 278.831,A -85,B 0,C 180,E1 -20065.959,E2 -20065.959} C_VEL
LIN {X 0,Y 243.989,Z 214.959,A -85,B 0,C 180,E1 -20067.933,E2 -20067.933} C_VEL
LIN {X 0,Y 237.656,Z 197.61,A -85,B 0,C 180,E1 -20069.269,E2 -20069.269} C_VEL
LIN {X 0,Y 230.899,Z 180.501,A -85,B 0,C 180,E1 -20070.73,E2 -20070.73} C_VEL
LIN {X 0,Y 228.69,Z 175.899,A -85,B 0,C 180,E1 -20071.191,E2 -20071.191} C_VEL
LIN {X 0,Y 228.526,Z 175.017,A -85,B 0,C 180,E1 -20071.267,E2 -20071.267} C_VEL
LIN {X 0,Y 228.308,Z 175.044,A -85,B 0,C 180,E1 -20077.073,E2 -20077.073} C_VEL
LIN {X 0,Y 228.143,Z 175.061,A -85,B 0,C 180,E1 -20080.651,E2 -20080.651} C_VEL
LIN {X 0,Y 228.016,Z 175.073,A -85,B 0,C 180,E1 -20086.105,E2 -20086.105} C_VEL
LIN {X 0,Y 227.915,Z 175.097,A -85,B 0,C 180,E1 -20089.828,E2 -20089.828} C_VEL
LIN {X 0,Y 227.862,Z 175.09,A -85,B 0,C 180,E1 -20093.639,E2 -20093.639} C_VEL
LIN {X 0,Y 227.847,Z 175.103,A -85,B 0,C 180,E1 -20097.56,E2 -20097.56} C_VEL
LIN {X 0,Y 227.858,Z 175.091,A -85,B 0,C 180,E1 -20101.624,E2 -20101.624} C_VEL
LIN {X 0,Y 227.882,Z 175.09,A -85,B 0,C 180,E1 -20105.872,E2 -20105.872} C_VEL
LIN {X 0,Y 227.804,Z 175.107,A -85,B 0,C 180,E1 -20110.382,E2 -20110.382} C_VEL
LIN {X 0,Y 227.812,Z 175.082,A -85,B 0,C 180,E1 -20115.199,E2 -20115.199} C_VEL
LIN {X 0,Y 227.802,Z 175.098,A -85,B 0,C 180,E1 -20119.618,E2 -20119.618} C_VEL
LIN {X 0,Y 227.868,Z 175.099,A -85,B 0,C 180,E1 -20124.126,E2 -20124.126} C_VEL
LIN {X 0,Y 227.858,Z 175.092,A -85,B 0,C 180,E1 -20128.376,E2 -20128.376} C_VEL
LIN {X 0,Y 227.857,Z 175.102,A -85,B 0,C 180,E1 -20132.441,E2 -20132.441} C_VEL
LIN {X 0,Y 227.892,Z 175.09,A -85,B 0,C 180,E1 -20136.365,E2 -20136.365} C_VEL
LIN {X 0,Y 227.893,Z 175.096,A -85,B 0,C 180,E1 -20140.17,E2 -20140.17} C_VEL
LIN {X 0,Y 228.011,Z 175.078,A -85,B 0,C 180,E1 -20143.894,E2 -20143.894} C_VEL
LIN {X 0,Y 228.143,Z 175.065,A -85,B 0,C 180,E1 -20149.349,E2 -20149.349} C_VEL
LIN {X 0,Y 228.309,Z 175.039,A -85,B 0,C 180,E1 -20152.927,E2 -20152.927} C_VEL
LIN {X 0,Y 228.537,Z 175.019,A -85,B 0,C 180,E1 -20158.238,E2 -20158.238} C_VEL
LIN {X 0,Y 228.537,Z 175.013,A -85,B 0,C 180,E1 -20161.762,E2 -20161.762} C_VEL
LIN {X 0,Y 228.302,Z 175.016,A -85,B 0,C 180,E1 -20167.073,E2 -20167.073} C_VEL
LIN {X 0,Y 228.126,Z 175.062,A -85,B 0,C 180,E1 -20170.652,E2 -20170.652} C_VEL
LIN {X 0,Y 228.009,Z 175.079,A -85,B 0,C 180,E1 -20176.106,E2 -20176.106} C_VEL
LIN {X 0,Y 227.92,Z 175.077,A -85,B 0,C 180,E1 -20181.717,E2 -20181.717} C_VEL
LIN {X 0,Y 227.903,Z 175.095,A -85,B 0,C 180,E1 -20186.581,E2 -20186.581} C_VEL
LIN {X 0,Y 227.871,Z 175.1,A -85,B 0,C 180,E1 -20190.279,E2 -20190.279} C_VEL
LIN {X 0,Y 227.878,Z 175.098,A -85,B 0,C 180,E1 -20193.72,E2 -20193.72} C_VEL
LIN {X 0,Y 227.869,Z 175.101,A -85,B 0,C 180,E1 -20196.857,E2 -20196.857} C_VEL
LIN {X 0,Y 227.142,Z 175.192,A -85,B 0,C 180,E1 -20198.332,E2 -20198.332} C_VEL
LIN {X 0,Y 224.274,Z 175.549,A -85,B 0,C 180,E1 -20200.74,E2 -20200.74} C_VEL
LIN {X 0,Y 221.868,Z 175.85,A -85,B 0,C 180,E1 -20202.704,E2 -20202.704} C_VEL
LIN {X 0,Y 220.834,Z 175.975,A -85,B 0,C 180,E1 -20204.229,E2 -20204.229} C_VEL
LIN {X 0,Y 220.746,Z 175.982,A -85,B 0,C 180,E1 -20204.746,E2 -20204.746} C_VEL
LIN {X 0,Y 220.749,Z 175.988,A -85,B 0,C 180,E1 -20208.042,E2 -20208.042} C_VEL
LIN {X 0,Y 220.873,Z 176.127,A -85,B 0,C 180,E1 -20211.623,E2 -20211.623} C_VEL
LIN {X 0,Y 222.765,Z 184.429,A -85,B 0,C 180,E1 -20215.397,E2 -20215.397} C_VEL
LIN {X 0,Y 223.148,Z 186.11,A -85,B 0,C 180,E1 -20216.066,E2 -20216.066} C_VEL
LIN {X 0,Y 231.252,Z 206.805,A -85,B 0,C 180,E1 -20217.904,E2 -20217.904} C_VEL
LIN {X 0,Y 233.701,Z 214.194,A -85,B 0,C 180,E1 -20218.471,E2 -20218.471} C_VEL
LIN {X 0,Y 236.851,Z 238.3,A -85,B 0,C 180,E1 -20219.706,E2 -20219.706} C_VEL
LIN {X 0,Y 234.514,Z 294.813,A -85,B 0,C 180,E1 -20221.531,E2 -20221.531} C_VEL
LIN {X 0,Y 233.352,Z 308.32,A -85,B 0,C 180,E1 -20222.293,E2 -20222.293} C_VEL
LIN {X 0,Y 231.845,Z 320.675,A -85,B 0,C 180,E1 -20223.319,E2 -20223.319} C_VEL
LIN {X 0,Y 229.996,Z 332.579,A -85,B 0,C 180,E1 -20224.672,E2 -20224.672} C_VEL
LIN {X 0,Y 227.909,Z 344.048,A -85,B 0,C 180,E1 -20226.367,E2 -20226.367} C_VEL
LIN {X 0,Y 225.907,Z 354.422,A -85,B 0,C 180,E1 -20228.319,E2 -20228.319} C_VEL
LIN {X 0,Y 224.02,Z 363.352,A -85,B 0,C 180,E1 -20230.422,E2 -20230.422} C_VEL
LIN {X 0,Y 222.539,Z 370.712,A -85,B 0,C 180,E1 -20232.541,E2 -20232.541} C_VEL
LIN {X 0,Y 220.939,Z 378.339,A -85,B 0,C 180,E1 -20235.257,E2 -20235.257} C_VEL
LIN {X 0,Y 219.764,Z 384.453,A -85,B 0,C 180,E1 -20238.002,E2 -20238.002} C_VEL
LIN {X 0,Y 219.065,Z 389.275,A -85,B 0,C 180,E1 -20240.769,E2 -20240.769} C_VEL
LIN {X 0,Y 218.649,Z 392.936,A -85,B 0,C 180,E1 -20243.541,E2 -20243.541} C_VEL
LIN {X 0,Y 218.521,Z 395.55,A -85,B 0,C 180,E1 -20246.312,E2 -20246.312} C_VEL
LIN {X 0,Y 218.567,Z 396.768,A -85,B 0,C 180,E1 -20248.157,E2 -20248.157} C_VEL
LIN {X 0,Y 218.648,Z 397.541,A -85,B 0,C 180,E1 -20250,E2 -20250} C_VEL
LIN {X 0,Y 218.552,Z 397.887,A -85,B 0,C 180,E1 -20251.843,E2 -20251.843} C_VEL
LIN {X 0,Y 218.569,Z 397.413,A -85,B 0,C 180,E1 -20255.536,E2 -20255.536} C_VEL
LIN {X 0,Y 218.762,Z 396.572,A -85,B 0,C 180,E1 -20257.383,E2 -20257.383} C_VEL
LIN {X 0,Y 219.655,Z 393.641,A -85,B 0,C 180,E1 -20261.068,E2 -20261.068} C_VEL
LIN {X 0,Y 220.776,Z 390.325,A -85,B 0,C 180,E1 -20263.813,E2 -20263.813} C_VEL
LIN {X 0,Y 222.462,Z 385.955,A -85,B 0,C 180,E1 -20266.519,E2 -20266.519} C_VEL
LIN {X 0,Y 225.079,Z 379.411,A -85,B 0,C 180,E1 -20269.613,E2 -20269.613} C_VEL
LIN {X 0,Y 227.555,Z 372.417,A -85,B 0,C 180,E1 -20272.183,E2 -20272.183} C_VEL
LIN {X 0,Y 230.716,Z 363.444,A -85,B 0,C 180,E1 -20274.762,E2 -20274.762} C_VEL
LIN {X 0,Y 234.079,Z 353.431,A -85,B 0,C 180,E1 -20277.008,E2 -20277.008} C_VEL
LIN {X 0,Y 237.086,Z 343.252,A -85,B 0,C 180,E1 -20278.797,E2 -20278.797} C_VEL
LIN {X 0,Y 240.053,Z 332.03,A -85,B 0,C 180,E1 -20280.333,E2 -20280.333} C_VEL
LIN {X 0,Y 242.307,Z 321.475,A -85,B 0,C 180,E1 -20281.472,E2 -20281.472} C_VEL
LIN {X 0,Y 244.349,Z 310.137,A -85,B 0,C 180,E1 -20282.391,E2 -20282.391} C_VEL
LIN {X 0,Y 246.129,Z 296.936,A -85,B 0,C 180,E1 -20283.131,E2 -20283.131} C_VEL
LIN {X 0,Y 247.369,Z 278.714,A -85,B 0,C 180,E1 -20283.767,E2 -20283.767} C_VEL
LIN {X 0,Y 249.399,Z 241.213,A -85,B 0,C 180,E1 -20284.927,E2 -20284.927} C_VEL
LIN {X 0,Y 247.846,Z 229.643,A -85,B 0,C 180,E1 -20285.743,E2 -20285.743} C_VEL
LIN {X 0,Y 243.382,Z 218.913,A -85,B 0,C 180,E1 -20287.199,E2 -20287.199} C_VEL
LIN {X 0,Y 238.269,Z 208.397,A -85,B 0,C 180,E1 -20288.933,E2 -20288.933} C_VEL
LIN {X 0,Y 232.827,Z 198.763,A -85,B 0,C 180,E1 -20290.863,E2 -20290.863} C_VEL
LIN {X 0,Y 229.634,Z 193.613,A -85,B 0,C 180,E1 -20292.074,E2 -20292.074} C_VEL
LIN {X 0,Y 226.54,Z 188.783,A -85,B 0,C 180,E1 -20293.308,E2 -20293.308} C_VEL
LIN {X 0,Y 223.53,Z 184.356,A -85,B 0,C 180,E1 -20294.579,E2 -20294.579} C_VEL
LIN {X 0,Y 223.09,Z 183.349,A -85,B 0,C 180,E1 -20294.87,E2 -20294.87} C_VEL
LIN {X 0,Y 221.621,Z 178.666,A -85,B 0,C 180,E1 -20298.245,E2 -20298.245} C_VEL
LIN {X 0,Y 220.791,Z 175.975,A -85,B 0,C 180,E1 -20300.46,E2 -20300.46} C_VEL
LIN {X 0,Y 220.826,Z 175.97,A -85,B 0,C 180,E1 -20302.793,E2 -20302.793} C_VEL
LIN {X 0,Y 220.813,Z 175.968,A -85,B 0,C 180,E1 -20307.243,E2 -20307.243} C_VEL
LIN {X 0,Y 220.796,Z 175.969,A -85,B 0,C 180,E1 -20311.481,E2 -20311.481} C_VEL
LIN {X 0,Y 220.797,Z 175.967,A -85,B 0,C 180,E1 -20315.557,E2 -20315.557} C_VEL
LIN {X 0,Y 220.847,Z 175.959,A -85,B 0,C 180,E1 -20319.51,E2 -20319.51} C_VEL
LIN {X 0,Y 220.968,Z 175.948,A -85,B 0,C 180,E1 -20323.366,E2 -20323.366} C_VEL
LIN {X 0,Y 221.051,Z 175.933,A -85,B 0,C 180,E1 -20329.003,E2 -20329.003} C_VEL
LIN {X 0,Y 221.247,Z 175.91,A -85,B 0,C 180,E1 -20332.7,E2 -20332.7} C_VEL
LIN {X 0,Y 221.468,Z 175.882,A -85,B 0,C 180,E1 -20338.182,E2 -20338.182} C_VEL
LIN {X 0,Y 221.468,Z 175.885,A -85,B 0,C 180,E1 -20341.819,E2 -20341.819} C_VEL
LIN {X 0,Y 221.244,Z 175.924,A -85,B 0,C 180,E1 -20347.3,E2 -20347.3} C_VEL
LIN {X 0,Y 221.053,Z 175.952,A -85,B 0,C 180,E1 -20350.997,E2 -20350.997} C_VEL
LIN {X 0,Y 221.047,Z 176.083,A -85,B 0,C 180,E1 -20351.927,E2 -20351.927} C_VEL
LIN {X 0,Y 221.254,Z 177.128,A -85,B 0,C 180,E1 -20352.614,E2 -20352.614} C_VEL
LIN {X 0,Y 222.538,Z 179.556,A -85,B 0,C 180,E1 -20353.237,E2 -20353.237} C_VEL
LIN {X 0,Y 225.424,Z 182.937,A -85,B 0,C 180,E1 -20354.443,E2 -20354.443} C_VEL
LIN {X 0,Y 229.51,Z 188.741,A -85,B 0,C 180,E1 -20356.079,E2 -20356.079} C_VEL
LIN {X 0,Y 235.335,Z 197.862,A -85,B 0,C 180,E1 -20358.24,E2 -20358.24} C_VEL
LIN {X 0,Y 239.765,Z 205.368,A -85,B 0,C 180,E1 -20359.755,E2 -20359.755} C_VEL
LIN {X 0,Y 245.084,Z 215.639,A -85,B 0,C 180,E1 -20361.497,E2 -20361.497} C_VEL
LIN {X 0,Y 250.062,Z 226.924,A -85,B 0,C 180,E1 -20363.06,E2 -20363.06} C_VEL
LIN {X 0,Y 249.179,Z 244.716,A -85,B 0,C 180,E1 -20363.63,E2 -20363.63} C_VEL
LIN {X 0,Y 246.747,Z 284.457,A -85,B 0,C 180,E1 -20364.877,E2 -20364.877} C_VEL
LIN {X 0,Y 245.173,Z 298.216,A -85,B 0,C 180,E1 -20365.629,E2 -20365.629} C_VEL
LIN {X 0,Y 243.495,Z 309.243,A -85,B 0,C 180,E1 -20366.522,E2 -20366.522} C_VEL
LIN {X 0,Y 241.116,Z 321.172,A -85,B 0,C 180,E1 -20367.799,E2 -20367.799} C_VEL
LIN {X 0,Y 238.121,Z 333.105,A -85,B 0,C 180,E1 -20369.464,E2 -20369.464} C_VEL
LIN {X 0,Y 235.281,Z 342.985,A -85,B 0,C 180,E1 -20371.234,E2 -20371.234} C_VEL
LIN {X 0,Y 232.613,Z 351.248,A -85,B 0,C 180,E1 -20373.074,E2 -20373.074} C_VEL
LIN {X 0,Y 229.414,Z 360.243,A -85,B 0,C 180,E1 -20375.596,E2 -20375.596} C_VEL
LIN {X 0,Y 226.456,Z 367.967,A -85,B 0,C 180,E1 -20378.367,E2 -20378.367} C_VEL
LIN {X 0,Y 223.97,Z 374.08,A -85,B 0,C 180,E1 -20381.221,E2 -20381.221} C_VEL
LIN {X 0,Y 221.983,Z 378.81,A -85,B 0,C 180,E1 -20384.149,E2 -20384.149} C_VEL
LIN {X 0,Y 220.428,Z 382.349,A -85,B 0,C 180,E1 -20387.166,E2 -20387.166} C_VEL
LIN {X 0,Y 219.294,Z 384.738,A -85,B 0,C 180,E1 -20390.279,E2 -20390.279} C_VEL
LIN {X 0,Y 218.533,Z 385.98,A -85,B 0,C 180,E1 -20393.514,E2 -20393.514} C_VEL
LIN {X 0,Y 218.173,Z 385.97,A -85,B 0,C 180,E1 -20396.881,E2 -20396.881} C_VEL
LIN {X 0,Y 218.217,Z 384.494,A -85,B 0,C 180,E1 -20400.41,E2 -20400.41} C_VEL
LIN {X 0,Y 218.783,Z 381.387,A -85,B 0,C 180,E1 -20404.087,E2 -20404.087} C_VEL
LIN {X 0,Y 219.561,Z 376.978,A -85,B 0,C 180,E1 -20407.411,E2 -20407.411} C_VEL
LIN {X 0,Y 220.567,Z 371.495,A -85,B 0,C 180,E1 -20410.454,E2 -20410.454} C_VEL
LIN {X 0,Y 222.031,Z 364.467,A -85,B 0,C 180,E1 -20413.448,E2 -20413.448} C_VEL
LIN {X 0,Y 223.758,Z 356.71,A -85,B 0,C 180,E1 -20416.031,E2 -20416.031} C_VEL
LIN {X 0,Y 225.525,Z 348.231,A -85,B 0,C 180,E1 -20418.313,E2 -20418.313} C_VEL
LIN {X 0,Y 227.587,Z 337.996,A -85,B 0,C 180,E1 -20420.526,E2 -20420.526} C_VEL
LIN {X 0,Y 229.477,Z 327.608,A -85,B 0,C 180,E1 -20422.3,E2 -20422.3} C_VEL
LIN {X 0,Y 231.353,Z 315.698,A -85,B 0,C 180,E1 -20423.897,E2 -20423.897} C_VEL
LIN {X 0,Y 232.926,Z 303.227,A -85,B 0,C 180,E1 -20425.167,E2 -20425.167} C_VEL
LIN {X 0,Y 234.228,Z 290.305,A -85,B 0,C 180,E1 -20426.087,E2 -20426.087} C_VEL
LIN {X 0,Y 235.103,Z 276.86,A -85,B 0,C 180,E1 -20426.699,E2 -20426.699} C_VEL
LIN {X 0,Y 237.547,Z 216.583,A -85,B 0,C 180,E1 -20428.596,E2 -20428.596} C_VEL
LIN {X 0,Y 230.764,Z 198.116,A -85,B 0,C 180,E1 -20430.081,E2 -20430.081} C_VEL
LIN {X 0,Y 225.183,Z 183.975,A -85,B 0,C 180,E1 -20431.339,E2 -20431.339} C_VEL
LIN {X 0,Y 221.499,Z 176.493,A -85,B 0,C 180,E1 -20432.131,E2 -20432.131} C_VEL
LIN {X 0,Y 221.381,Z 175.91,A -85,B 0,C 180,E1 -20432.217,E2 -20432.217} C_VEL
LIN {X 0,Y 221.246,Z 175.924,A -85,B 0,C 180,E1 -20437.3,E2 -20437.3} C_VEL
LIN {X 0,Y 221.062,Z 175.941,A -85,B 0,C 180,E1 -20440.997,E2 -20440.997} C_VEL
LIN {X 0,Y 220.976,Z 175.946,A -85,B 0,C 180,E1 -20446.633,E2 -20446.633} C_VEL
LIN {X 0,Y 220.87,Z 175.973,A -85,B 0,C 180,E1 -20450.488,E2 -20450.488} C_VEL
LIN {X 0,Y 220.8,Z 175.968,A -85,B 0,C 180,E1 -20454.443,E2 -20454.443} C_VEL
LIN {X 0,Y 220.801,Z 175.98,A -85,B 0,C 180,E1 -20458.519,E2 -20458.519} C_VEL
LIN {X 0,Y 220.814,Z 175.962,A -85,B 0,C 180,E1 -20462.757,E2 -20462.757} C_VEL
LIN {X 0,Y 220.811,Z 175.975,A -85,B 0,C 180,E1 -20467.278,E2 -20467.278} C_VEL
LIN {X 0,Y 220.751,Z 175.981,A -85,B 0,C 180,E1 -20471.957,E2 -20471.957} C_VEL
LIN {X 0,Y 220.754,Z 175.956,A -85,B 0,C 180,E1 -20475.541,E2 -20475.541} C_VEL
LIN {X 0,Y 220.783,Z 175.974,A -85,B 0,C 180,E1 -20480.458,E2 -20480.458} C_VEL
LIN {X 0,Y 220.827,Z 175.976,A -85,B 0,C 180,E1 -20482.793,E2 -20482.793} C_VEL
LIN {X 0,Y 220.814,Z 175.97,A -85,B 0,C 180,E1 -20487.243,E2 -20487.243} C_VEL
LIN {X 0,Y 220.806,Z 175.979,A -85,B 0,C 180,E1 -20491.482,E2 -20491.482} C_VEL
LIN {X 0,Y 220.847,Z 175.967,A -85,B 0,C 180,E1 -20495.562,E2 -20495.562} C_VEL
LIN {X 0,Y 220.852,Z 175.972,A -85,B 0,C 180,E1 -20499.51,E2 -20499.51} C_VEL
LIN {X 0,Y 220.972,Z 175.954,A -85,B 0,C 180,E1 -20503.367,E2 -20503.367} C_VEL
LIN {X 0,Y 221.062,Z 175.947,A -85,B 0,C 180,E1 -20509.003,E2 -20509.003} C_VEL
LIN {X 0,Y 221.246,Z 175.919,A -85,B 0,C 180,E1 -20512.7,E2 -20512.7} C_VEL
LIN {X 0,Y 221.471,Z 175.899,A -85,B 0,C 180,E1 -20518.181,E2 -20518.181} C_VEL
LIN {X 0,Y 221.47,Z 175.891,A -85,B 0,C 180,E1 -20521.818,E2 -20521.818} C_VEL
LIN {X 0,Y 221.239,Z 175.894,A -85,B 0,C 180,E1 -20527.3,E2 -20527.3} C_VEL
LIN {X 0,Y 221.048,Z 175.943,A -85,B 0,C 180,E1 -20530.997,E2 -20530.997} C_VEL
LIN {X 0,Y 220.971,Z 175.954,A -85,B 0,C 180,E1 -20536.633,E2 -20536.633} C_VEL
LIN {X 0,Y 220.847,Z 175.951,A -85,B 0,C 180,E1 -20540.491,E2 -20540.491} C_VEL
LIN {X 0,Y 220.804,Z 175.978,A -85,B 0,C 180,E1 -20544.442,E2 -20544.442} C_VEL
LIN {X 0,Y 220.797,Z 175.976,A -85,B 0,C 180,E1 -20548.519,E2 -20548.519} C_VEL
LIN {X 0,Y 220.813,Z 175.98,A -85,B 0,C 180,E1 -20552.757,E2 -20552.757} C_VEL
LIN {X 0,Y 220.803,Z 175.983,A -85,B 0,C 180,E1 -20557.275,E2 -20557.275} C_VEL
LIN {X 0,Y 220.749,Z 175.987,A -85,B 0,C 180,E1 -20561.957,E2 -20561.957} C_VEL
LIN {X 0,Y 220.746,Z 175.982,A -85,B 0,C 180,E1 -20564.746,E2 -20564.746} C_VEL
LIN {X 0,Y 220.054,Z 176.067,A -85,B 0,C 180,E1 -20565.76,E2 -20565.76} C_VEL
LIN {X 0,Y 217.196,Z 176.431,A -85,B 0,C 180,E1 -20567.354,E2 -20567.354} C_VEL
LIN {X 0,Y 214.36,Z 176.779,A -85,B 0,C 180,E1 -20568.988,E2 -20568.988} C_VEL
LIN {X 0,Y 213.738,Z 176.855,A -85,B 0,C 180,E1 -20570.048,E2 -20570.048} C_VEL
LIN {X 0,Y 213.788,Z 176.912,A -85,B 0,C 180,E1 -20570.879,E2 -20570.879} C_VEL
LIN {X 0,Y 215.827,Z 185.714,A -85,B 0,C 180,E1 -20575.03,E2 -20575.03} C_VEL
LIN {X 0,Y 224.434,Z 207.432,A -85,B 0,C 180,E1 -20577.071,E2 -20577.071} C_VEL
LIN {X 0,Y 227.468,Z 216.402,A -85,B 0,C 180,E1 -20577.802,E2 -20577.802} C_VEL
LIN {X 0,Y 230.387,Z 239.043,A -85,B 0,C 180,E1 -20579.005,E2 -20579.005} C_VEL
LIN {X 0,Y 228.021,Z 294.296,A -85,B 0,C 180,E1 -20580.832,E2 -20580.832} C_VEL
LIN {X 0,Y 226.803,Z 307.893,A -85,B 0,C 180,E1 -20581.61,E2 -20581.61} C_VEL
LIN {X 0,Y 225.347,Z 319.759,A -85,B 0,C 180,E1 -20582.612,E2 -20582.612} C_VEL
LIN {X 0,Y 223.6,Z 331.078,A -85,B 0,C 180,E1 -20583.894,E2 -20583.894} C_VEL
LIN {X 0,Y 221.324,Z 342.767,A -85,B 0,C 180,E1 -20585.619,E2 -20585.619} C_VEL
LIN {X 0,Y 219.248,Z 353.34,A -85,B 0,C 180,E1 -20587.626,E2 -20587.626} C_VEL
LIN {X 0,Y 217.47,Z 361.67,A -85,B 0,C 180,E1 -20589.586,E2 -20589.586} C_VEL
LIN {X 0,Y 215.751,Z 369.945,A -85,B 0,C 180,E1 -20591.973,E2 -20591.973} C_VEL
LIN {X 0,Y 214.059,Z 377.682,A -85,B 0,C 180,E1 -20594.772,E2 -20594.772} C_VEL
LIN {X 0,Y 212.782,Z 383.882,A -85,B 0,C 180,E1 -20597.603,E2 -20597.603} C_VEL
LIN {X 0,Y 212.037,Z 388.786,A -85,B 0,C 180,E1 -20600.461,E2 -20600.461} C_VEL
LIN {X 0,Y 211.577,Z 392.522,A -85,B 0,C 180,E1 -20603.324,E2 -20603.324} C_VEL
LIN {X 0,Y 211.437,Z 395.206,A -85,B 0,C 180,E1 -20606.188,E2 -20606.188} C_VEL
LIN {X 0,Y 211.467,Z 396.457,A -85,B 0,C 180,E1 -20608.095,E2 -20608.095} C_VEL
LIN {X 0,Y 211.563,Z 397.293,A -85,B 0,C 180,E1 -20610,E2 -20610} C_VEL
LIN {X 0,Y 211.452,Z 397.674,A -85,B 0,C 180,E1 -20611.905,E2 -20611.905} C_VEL
LIN {X 0,Y 211.419,Z 397.615,A -85,B 0,C 180,E1 -20614.241,E2 -20614.241} C_VEL
LIN {X 0,Y 211.691,Z 396.476,A -85,B 0,C 180,E1 -20617.631,E2 -20617.631} C_VEL
LIN {X 0,Y 212.679,Z 393.622,A -85,B 0,C 180,E1 -20621.436,E2 -20621.436} C_VEL
LIN {X 0,Y 213.847,Z 390.389,A -85,B 0,C 180,E1 -20624.27,E2 -20624.27} C_VEL
LIN {X 0,Y 215.648,Z 386.111,A -85,B 0,C 180,E1 -20627.056,E2 -20627.056} C_VEL
LIN {X 0,Y 218.378,Z 379.66,A -85,B 0,C 180,E1 -20630.241,E2 -20630.241} C_VEL
LIN {X 0,Y 221.046,Z 372.669,A -85,B 0,C 180,E1 -20632.922,E2 -20632.922} C_VEL
LIN {X 0,Y 224.31,Z 363.952,A -85,B 0,C 180,E1 -20635.519,E2 -20635.519} C_VEL
LIN {X 0,Y 227.494,Z 355.059,A -85,B 0,C 180,E1 -20637.607,E2 -20637.607} C_VEL
LIN {X 0,Y 230.946,Z 344.188,A -85,B 0,C 180,E1 -20639.638,E2 -20639.638} C_VEL
LIN {X 0,Y 234.019,Z 333.26,A -85,B 0,C 180,E1 -20641.202,E2 -20641.202} C_VEL
LIN {X 0,Y 236.775,Z 321.166,A -85,B 0,C 180,E1 -20642.547,E2 -20642.547} C_VEL
LIN {X 0,Y 239.141,Z 308.514,A -85,B 0,C 180,E1 -20643.565,E2 -20643.565} C_VEL
LIN {X 0,Y 240.878,Z 294.968,A -85,B 0,C 180,E1 -20644.304,E2 -20644.304} C_VEL
LIN {X 0,Y 242.582,Z 268.747,A -85,B 0,C 180,E1 -20645.17,E2 -20645.17} C_VEL
LIN {X 0,Y 244.074,Z 242.307,A -85,B 0,C 180,E1 -20646.005,E2 -20646.005} C_VEL
LIN {X 0,Y 242.843,Z 232.653,A -85,B 0,C 180,E1 -20646.704,E2 -20646.704} C_VEL
LIN {X 0,Y 238.51,Z 222.081,A -85,B 0,C 180,E1 -20648.217,E2 -20648.217} C_VEL
LIN {X 0,Y 233.601,Z 212.015,A -85,B 0,C 180,E1 -20649.978,E2 -20649.978} C_VEL
LIN {X 0,Y 228.954,Z 203.635,A -85,B 0,C 180,E1 -20651.74,E2 -20651.74} C_VEL
LIN {X 0,Y 225.941,Z 198.625,A -85,B 0,C 180,E1 -20652.948,E2 -20652.948} C_VEL
LIN {X 0,Y 223.015,Z 194.027,A -85,B 0,C 180,E1 -20654.18,E2 -20654.18} C_VEL
LIN {X 0,Y 219.44,Z 188.623,A -85,B 0,C 180,E1 -20655.798,E2 -20655.798} C_VEL
LIN {X 0,Y 215.914,Z 183.603,A -85,B 0,C 180,E1 -20657.514,E2 -20657.514} C_VEL
LIN {X 0,Y 215.635,Z 182.944,A -85,B 0,C 180,E1 -20657.763,E2 -20657.763} C_VEL
LIN {X 0,Y 214.696,Z 179.759,A -85,B 0,C 180,E1 -20660.333,E2 -20660.333} C_VEL
LIN {X 0,Y 213.765,Z 176.848,A -85,B 0,C 180,E1 -20663.074,E2 -20663.074} C_VEL
LIN {X 0,Y 213.756,Z 176.851,A -85,B 0,C 180,E1 -20666.018,E2 -20666.018} C_VEL
LIN {X 0,Y 213.748,Z 176.846,A -85,B 0,C 180,E1 -20670.449,E2 -20670.449} C_VEL
LIN {X 0,Y 213.747,Z 176.845,A -85,B 0,C 180,E1 -20674.695,E2 -20674.695} C_VEL
LIN {X 0,Y 213.776,Z 176.842,A -85,B 0,C 180,E1 -20678.8,E2 -20678.8} C_VEL
LIN {X 0,Y 213.88,Z 176.836,A -85,B 0,C 180,E1 -20682.798,E2 -20682.798} C_VEL
LIN {X 0,Y 213.911,Z 176.839,A -85,B 0,C 180,E1 -20686.704,E2 -20686.704} C_VEL
LIN {X 0,Y 214.128,Z 176.805,A -85,B 0,C 180,E1 -20690.555,E2 -20690.555} C_VEL
LIN {X 0,Y 214.186,Z 176.791,A -85,B 0,C 180,E1 -20692.458,E2 -20692.458} C_VEL
LIN {X 0,Y 214.405,Z 176.762,A -85,B 0,C 180,E1 -20698.122,E2 -20698.122} C_VEL
LIN {X 0,Y 214.515,Z 176.763,A -85,B 0,C 180,E1 -20700,E2 -20700} C_VEL
LIN {X 0,Y 214.405,Z 176.764,A -85,B 0,C 180,E1 -20701.879,E2 -20701.879} C_VEL
LIN {X 0,Y 214.165,Z 176.802,A -85,B 0,C 180,E1 -20708.492,E2 -20708.492} C_VEL
LIN {X 0,Y 214.171,Z 176.933,A -85,B 0,C 180,E1 -20709.444,E2 -20709.444} C_VEL
LIN {X 0,Y 214.274,Z 177.594,A -85,B 0,C 180,E1 -20709.819,E2 -20709.819} C_VEL
LIN {X 0,Y 215.366,Z 180.098,A -85,B 0,C 180,E1 -20710.475,E2 -20710.475} C_VEL
LIN {X 0,Y 217.595,Z 182.17,A -85,B 0,C 180,E1 -20711.528,E2 -20711.528} C_VEL
LIN {X 0,Y 220.216,Z 186.145,A -85,B 0,C 180,E1 -20712.792,E2 -20712.792} C_VEL
LIN {X 0,Y 222.206,Z 188.516,A -85,B 0,C 180,E1 -20713.664,E2 -20713.664} C_VEL
LIN {X 0,Y 226.152,Z 194.28,A -85,B 0,C 180,E1 -20715.331,E2 -20715.331} C_VEL
LIN {X 0,Y 231.688,Z 203.117,A -85,B 0,C 180,E1 -20717.493,E2 -20717.493} C_VEL
LIN {X 0,Y 236.708,Z 211.972,A -85,B 0,C 180,E1 -20719.297,E2 -20719.297} C_VEL
LIN {X 0,Y 242.187,Z 223.237,A -85,B 0,C 180,E1 -20721.181,E2 -20721.181} C_VEL
LIN {X 0,Y 244.753,Z 229.284,A -85,B 0,C 180,E1 -20722.028,E2 -20722.028} C_VEL
LIN {X 0,Y 241.403,Z 284.264,A -85,B 0,C 180,E1 -20723.777,E2 -20723.777} C_VEL
LIN {X 0,Y 239.769,Z 298.105,A -85,B 0,C 180,E1 -20724.535,E2 -20724.535} C_VEL
LIN {X 0,Y 237.927,Z 309.641,A -85,B 0,C 180,E1 -20725.476,E2 -20725.476} C_VEL
LIN {X 0,Y 235.54,Z 321.073,A -85,B 0,C 180,E1 -20726.719,E2 -20726.719} C_VEL
LIN {X 0,Y 232.557,Z 332.542,A -85,B 0,C 180,E1 -20728.336,E2 -20728.336} C_VEL
LIN {X 0,Y 229.536,Z 342.526,A -85,B 0,C 180,E1 -20730.128,E2 -20730.128} C_VEL
LIN {X 0,Y 226.352,Z 351.901,A -85,B 0,C 180,E1 -20732.254,E2 -20732.254} C_VEL
LIN {X 0,Y 223.43,Z 359.743,A -85,B 0,C 180,E1 -20734.485,E2 -20734.485} C_VEL
LIN {X 0,Y 220.241,Z 367.61,A -85,B 0,C 180,E1 -20737.323,E2 -20737.323} C_VEL
LIN {X 0,Y 217.555,Z 373.867,A -85,B 0,C 180,E1 -20740.248,E2 -20740.248} C_VEL
LIN {X 0,Y 215.371,Z 378.709,A -85,B 0,C 180,E1 -20743.257,E2 -20743.257} C_VEL
LIN {X 0,Y 213.654,Z 382.323,A -85,B 0,C 180,E1 -20746.359,E2 -20746.359} C_VEL
LIN {X 0,Y 212.399,Z 384.786,A -85,B 0,C 180,E1 -20749.556,E2 -20749.556} C_VEL
LIN {X 0,Y 211.471,Z 386.201,A -85,B 0,C 180,E1 -20753.258,E2 -20753.258} C_VEL
LIN {X 0,Y 211.118,Z 386.219,A -85,B 0,C 180,E1 -20756.329,E2 -20756.329} C_VEL
LIN {X 0,Y 211.112,Z 384.848,A -85,B 0,C 180,E1 -20760.042,E2 -20760.042} C_VEL
LIN {X 0,Y 211.632,Z 381.955,A -85,B 0,C 180,E1 -20763.72,E2 -20763.72} C_VEL
LIN {X 0,Y 212.275,Z 378.538,A -85,B 0,C 180,E1 -20766.59,E2 -20766.59} C_VEL
LIN {X 0,Y 213.169,Z 373.495,A -85,B 0,C 180,E1 -20769.746,E2 -20769.746} C_VEL
LIN {X 0,Y 214.541,Z 366.91,A -85,B 0,C 180,E1 -20772.853,E2 -20772.853} C_VEL
LIN {X 0,Y 216.359,Z 358.988,A -85,B 0,C 180,E1 -20775.77,E2 -20775.77} C_VEL
LIN {X 0,Y 218.357,Z 349.94,A -85,B 0,C 180,E1 -20778.395,E2 -20778.395} C_VEL
LIN {X 0,Y 220.368,Z 340.42,A -85,B 0,C 180,E1 -20780.593,E2 -20780.593} C_VEL
LIN {X 0,Y 222.379,Z 330.065,A -85,B 0,C 180,E1 -20782.509,E2 -20782.509} C_VEL
LIN {X 0,Y 224.286,Z 318.819,A -85,B 0,C 180,E1 -20784.155,E2 -20784.155} C_VEL
LIN {X 0,Y 225.891,Z 307.169,A -85,B 0,C 180,E1 -20785.463,E2 -20785.463} C_VEL
LIN {X 0,Y 227.38,Z 293.816,A -85,B 0,C 180,E1 -20786.555,E2 -20786.555} C_VEL
LIN {X 0,Y 228.434,Z 280.332,A -85,B 0,C 180,E1 -20787.264,E2 -20787.264} C_VEL
LIN {X 0,Y 231.065,Z 218.034,A -85,B 0,C 180,E1 -20789.296,E2 -20789.296} C_VEL
LIN {X 0,Y 221.749,Z 192.759,A -85,B 0,C 180,E1 -20791.455,E2 -20791.455} C_VEL
LIN {X 0,Y 217.411,Z 183.273,A -85,B 0,C 180,E1 -20792.435,E2 -20792.435} C_VEL
LIN {X 0,Y 214.462,Z 178.075,A -85,B 0,C 180,E1 -20793.079,E2 -20793.079} C_VEL
LIN {X 0,Y 214.174,Z 176.803,A -85,B 0,C 180,E1 -20793.234,E2 -20793.234} C_VEL
LIN {X 0,Y 214.187,Z 176.804,A -85,B 0,C 180,E1 -20797.542,E2 -20797.542} C_VEL
LIN {X 0,Y 213.992,Z 176.821,A -85,B 0,C 180,E1 -20801.365,E2 -20801.365} C_VEL
LIN {X 0,Y 213.88,Z 176.841,A -85,B 0,C 180,E1 -20805.241,E2 -20805.241} C_VEL
LIN {X 0,Y 213.812,Z 176.851,A -85,B 0,C 180,E1 -20809.19,E2 -20809.19} C_VEL
LIN {X 0,Y 213.766,Z 176.846,A -85,B 0,C 180,E1 -20813.237,E2 -20813.237} C_VEL
LIN {X 0,Y 213.786,Z 176.853,A -85,B 0,C 180,E1 -20817.427,E2 -20817.427} C_VEL
LIN {X 0,Y 213.76,Z 176.845,A -85,B 0,C 180,E1 -20821.739,E2 -20821.739} C_VEL
LIN {X 0,Y 213.746,Z 176.853,A -85,B 0,C 180,E1 -20826.288,E2 -20826.288} C_VEL
LIN {X 0,Y 213.7,Z 176.864,A -85,B 0,C 180,E1 -20831.128,E2 -20831.128} C_VEL
LIN {X 0,Y 213.703,Z 176.849,A -85,B 0,C 180,E1 -20833.68,E2 -20833.68} C_VEL
LIN {X 0,Y 213.702,Z 176.83,A -85,B 0,C 180,E1 -20836.346,E2 -20836.346} C_VEL
LIN {X 0,Y 213.706,Z 176.86,A -85,B 0,C 180,E1 -20841.329,E2 -20841.329} C_VEL
LIN {X 0,Y 213.756,Z 176.854,A -85,B 0,C 180,E1 -20846.018,E2 -20846.018} C_VEL
LIN {X 0,Y 213.752,Z 176.855,A -85,B 0,C 180,E1 -20850.449,E2 -20850.449} C_VEL
LIN {X 0,Y 213.783,Z 176.851,A -85,B 0,C 180,E1 -20854.699,E2 -20854.699} C_VEL
LIN {X 0,Y 213.779,Z 176.852,A -85,B 0,C 180,E1 -20858.8,E2 -20858.8} C_VEL
LIN {X 0,Y 213.881,Z 176.84,A -85,B 0,C 180,E1 -20862.798,E2 -20862.798} C_VEL
LIN {X 0,Y 213.919,Z 176.831,A -85,B 0,C 180,E1 -20866.704,E2 -20866.704} C_VEL
LIN {X 0,Y 214.139,Z 176.811,A -85,B 0,C 180,E1 -20870.555,E2 -20870.555} C_VEL
LIN {X 0,Y 214.079,Z 176.809,A -85,B 0,C 180,E1 -20874.348,E2 -20874.348} C_VEL
LIN {X 0,Y 214.408,Z 176.778,A -85,B 0,C 180,E1 -20878.121,E2 -20878.121} C_VEL
LIN {X 0,Y 214.515,Z 176.764,A -85,B 0,C 180,E1 -20880,E2 -20880} C_VEL
LIN {X 0,Y 214.407,Z 176.77,A -85,B 0,C 180,E1 -20881.878,E2 -20881.878} C_VEL
LIN {X 0,Y 214.18,Z 176.773,A -85,B 0,C 180,E1 -20887.542,E2 -20887.542} C_VEL
LIN {X 0,Y 213.98,Z 176.824,A -85,B 0,C 180,E1 -20891.365,E2 -20891.365} C_VEL
LIN {X 0,Y 213.871,Z 176.843,A -85,B 0,C 180,E1 -20895.241,E2 -20895.241} C_VEL
LIN {X 0,Y 213.791,Z 176.833,A -85,B 0,C 180,E1 -20899.192,E2 -20899.192} C_VEL
LIN {X 0,Y 213.786,Z 176.846,A -85,B 0,C 180,E1 -20903.234,E2 -20903.234} C_VEL
LIN {X 0,Y 213.786,Z 176.853,A -85,B 0,C 180,E1 -20907.426,E2 -20907.426} C_VEL
LIN {X 0,Y 213.76,Z 176.86,A -85,B 0,C 180,E1 -20911.739,E2 -20911.739} C_VEL
LIN {X 0,Y 213.743,Z 176.861,A -85,B 0,C 180,E1 -20916.289,E2 -20916.289} C_VEL
LIN {X 0,Y 213.699,Z 176.864,A -85,B 0,C 180,E1 -20921.128,E2 -20921.128} C_VEL
LIN {X 0,Y 213.648,Z 176.862,A -85,B 0,C 180,E1 -20924.737,E2 -20924.737} C_VEL
LIN {X 0,Y 213.704,Z 176.859,A -85,B 0,C 180,E1 -20929.147,E2 -20929.147} C_VEL
LIN {X 0,Y 213.738,Z 176.855,A -85,B 0,C 180,E1 -20930.048,E2 -20930.048} C_VEL
LIN {X 0,Y 213.371,Z 177.62,A -85,B 0,C 180,E1 -20930.967,E2 -20930.967} C_VEL
LIN {X 0,Y 212.455,Z 179.42,A -85,B 0,C 180,E1 -20931.793,E2 -20931.793} C_VEL
LIN {X 0,Y 210.739,Z 182.772,A -85,B 0,C 180,E1 -20932.947,E2 -20932.947} C_VEL
LIN {X 0,Y 209.852,Z 186.308,A -85,B 0,C 180,E1 -20933.8,E2 -20933.8} C_VEL
LIN {X 0,Y 210.083,Z 189.111,A -85,B 0,C 180,E1 -20934.287,E2 -20934.287} C_VEL
LIN {X 0,Y 210.486,Z 190.26,A -85,B 0,C 180,E1 -20934.433,E2 -20934.433} C_VEL
LIN {X 0,Y 217.835,Z 208.488,A -85,B 0,C 180,E1 -20936.235,E2 -20936.235} C_VEL
LIN {X 0,Y 221.28,Z 218.494,A -85,B 0,C 180,E1 -20937.092,E2 -20937.092} C_VEL
LIN {X 0,Y 223.927,Z 240.336,A -85,B 0,C 180,E1 -20938.28,E2 -20938.28} C_VEL
LIN {X 0,Y 221.482,Z 294.872,A -85,B 0,C 180,E1 -20940.146,E2 -20940.146} C_VEL
LIN {X 0,Y 220.139,Z 308.962,A -85,B 0,C 180,E1 -20940.996,E2 -20940.996} C_VEL
LIN {X 0,Y 218.543,Z 320.996,A -85,B 0,C 180,E1 -20942.075,E2 -20942.075} C_VEL
LIN {X 0,Y 216.581,Z 332.739,A -85,B 0,C 180,E1 -20943.501,E2 -20943.501} C_VEL
LIN {X 0,Y 214.35,Z 344.108,A -85,B 0,C 180,E1 -20945.289,E2 -20945.289} C_VEL
LIN {X 0,Y 212.221,Z 354.388,A -85,B 0,C 180,E1 -20947.357,E2 -20947.357} C_VEL
LIN {X 0,Y 210.125,Z 363.482,A -85,B 0,C 180,E1 -20949.652,E2 -20949.652} C_VEL
LIN {X 0,Y 208.611,Z 370.569,A -85,B 0,C 180,E1 -20951.843,E2 -20951.843} C_VEL
LIN {X 0,Y 206.898,Z 378.155,A -85,B 0,C 180,E1 -20954.737,E2 -20954.737} C_VEL
LIN {X 0,Y 205.489,Z 385.135,A -85,B 0,C 180,E1 -20958.158,E2 -20958.158} C_VEL
LIN {X 0,Y 204.804,Z 389.712,A -85,B 0,C 180,E1 -20961.117,E2 -20961.117} C_VEL
LIN {X 0,Y 204.437,Z 393.162,A -85,B 0,C 180,E1 -20964.08,E2 -20964.08} C_VEL
LIN {X 0,Y 204.342,Z 394.862,A -85,B 0,C 180,E1 -20966.056,E2 -20966.056} C_VEL
LIN {X 0,Y 204.37,Z 396.147,A -85,B 0,C 180,E1 -20968.029,E2 -20968.029} C_VEL
LIN {X 0,Y 204.48,Z 397.027,A -85,B 0,C 180,E1 -20970,E2 -20970} C_VEL
LIN {X 0,Y 204.355,Z 397.461,A -85,B 0,C 180,E1 -20971.971,E2 -20971.971} C_VEL
LIN {X 0,Y 204.347,Z 397.46,A -85,B 0,C 180,E1 -20974.144,E2 -20974.144} C_VEL
LIN {X 0,Y 204.643,Z 396.369,A -85,B 0,C 180,E1 -20977.896,E2 -20977.896} C_VEL
LIN {X 0,Y 205.075,Z 395.215,A -85,B 0,C 180,E1 -20979.867,E2 -20979.867} C_VEL
LIN {X 0,Y 206.063,Z 392.703,A -85,B 0,C 180,E1 -20982.808,E2 -20982.808} C_VEL
LIN {X 0,Y 207.485,Z 389.203,A -85,B 0,C 180,E1 -20985.723,E2 -20985.723} C_VEL
LIN {X 0,Y 209.641,Z 384.637,A -85,B 0,C 180,E1 -20988.571,E2 -20988.571} C_VEL
LIN {X 0,Y 212.104,Z 378.884,A -85,B 0,C 180,E1 -20991.376,E2 -20991.376} C_VEL
LIN {X 0,Y 215.061,Z 371.729,A -85,B 0,C 180,E1 -20994.11,E2 -20994.11} C_VEL
LIN {X 0,Y 218.574,Z 362.891,A -85,B 0,C 180,E1 -20996.754,E2 -20996.754} C_VEL
LIN {X 0,Y 222.355,Z 352.863,A -85,B 0,C 180,E1 -20999.076,E2 -20999.076} C_VEL
LIN {X 0,Y 225.656,Z 342.683,A -85,B 0,C 180,E1 -21000.924,E2 -21000.924} C_VEL
LIN {X 0,Y 228.829,Z 331.476,A -85,B 0,C 180,E1 -21002.512,E2 -21002.512} C_VEL
LIN {X 0,Y 231.344,Z 320.912,A -85,B 0,C 180,E1 -21003.671,E2 -21003.671} C_VEL
LIN {X 0,Y 233.784,Z 308.244,A -85,B 0,C 180,E1 -21004.702,E2 -21004.702} C_VEL
LIN {X 0,Y 235.602,Z 294.574,A -85,B 0,C 180,E1 -21005.452,E2 -21005.452} C_VEL
LIN {X 0,Y 237.678,Z 263.445,A -85,B 0,C 180,E1 -21006.484,E2 -21006.484} C_VEL
LIN {X 0,Y 238.892,Z 243.692,A -85,B 0,C 180,E1 -21007.11,E2 -21007.11} C_VEL
LIN {X 0,Y 237.904,Z 235.745,A -85,B 0,C 180,E1 -21007.719,E2 -21007.719} C_VEL
LIN {X 0,Y 234.303,Z 226.675,A -85,B 0,C 180,E1 -21009.062,E2 -21009.062} C_VEL
LIN {X 0,Y 229.733,Z 216.982,A -85,B 0,C 180,E1 -21010.798,E2 -21010.798} C_VEL
LIN {X 0,Y 224.978,Z 208.149,A -85,B 0,C 180,E1 -21012.723,E2 -21012.723} C_VEL
LIN {X 0,Y 221.625,Z 202.563,A -85,B 0,C 180,E1 -21014.149,E2 -21014.149} C_VEL
LIN {X 0,Y 219.586,Z 199.282,A -85,B 0,C 180,E1 -21015.078,E2 -21015.078} C_VEL
LIN {X 0,Y 216.171,Z 194.028,A -85,B 0,C 180,E1 -21016.712,E2 -21016.712} C_VEL
LIN {X 0,Y 212.174,Z 188.227,A -85,B 0,C 180,E1 -21018.807,E2 -21018.807} C_VEL
LIN {X 0,Y 209.232,Z 184.259,A -85,B 0,C 180,E1 -21020.508,E2 -21020.508} C_VEL
LIN {X 0,Y 208.229,Z 182.541,A -85,B 0,C 180,E1 -21021.221,E2 -21021.221} C_VEL
LIN {X 0,Y 206.72,Z 177.726,A -85,B 0,C 180,E1 -21026.171,E2 -21026.171} C_VEL
LIN {X 0,Y 206.696,Z 177.734,A -85,B 0,C 180,E1 -21029.335,E2 -21029.335} C_VEL
LIN {X 0,Y 206.685,Z 177.731,A -85,B 0,C 180,E1 -21033.766,E2 -21033.766} C_VEL
LIN {X 0,Y 206.708,Z 177.729,A -85,B 0,C 180,E1 -21038.038,E2 -21038.038} C_VEL
LIN {X 0,Y 206.805,Z 177.724,A -85,B 0,C 180,E1 -21042.191,E2 -21042.191} C_VEL
LIN {X 0,Y 206.852,Z 177.717,A -85,B 0,C 180,E1 -21046.241,E2 -21046.241} C_VEL
LIN {X 0,Y 207.074,Z 177.679,A -85,B 0,C 180,E1 -21050.23,E2 -21050.23} C_VEL
LIN {X 0,Y 207.041,Z 177.678,A -85,B 0,C 180,E1 -21054.155,E2 -21054.155} C_VEL
LIN {X 0,Y 207.345,Z 177.641,A -85,B 0,C 180,E1 -21058.058,E2 -21058.058} C_VEL
LIN {X 0,Y 207.483,Z 177.639,A -85,B 0,C 180,E1 -21060,E2 -21060} C_VEL
LIN {X 0,Y 207.345,Z 177.643,A -85,B 0,C 180,E1 -21061.943,E2 -21061.943} C_VEL
LIN {X 0,Y 207.049,Z 177.732,A -85,B 0,C 180,E1 -21066.273,E2 -21066.273} C_VEL
LIN {X 0,Y 207.942,Z 180.265,A -85,B 0,C 180,E1 -21066.977,E2 -21066.977} C_VEL
LIN {X 0,Y 210.171,Z 182.672,A -85,B 0,C 180,E1 -21068.292,E2 -21068.292} C_VEL
LIN {X 0,Y 211.425,Z 183.604,A -85,B 0,C 180,E1 -21068.964,E2 -21068.964} C_VEL
LIN {X 0,Y 213.205,Z 186.742,A -85,B 0,C 180,E1 -21070.004,E2 -21070.004} C_VEL
LIN {X 0,Y 215.301,Z 188.938,A -85,B 0,C 180,E1 -21071.056,E2 -21071.056} C_VEL
LIN {X 0,Y 217.597,Z 192.334,A -85,B 0,C 180,E1 -21072.193,E2 -21072.193} C_VEL
LIN {X 0,Y 219.285,Z 194.436,A -85,B 0,C 180,E1 -21072.965,E2 -21072.965} C_VEL
LIN {X 0,Y 223.198,Z 200.414,A -85,B 0,C 180,E1 -21074.717,E2 -21074.717} C_VEL
LIN {X 0,Y 227.76,Z 207.775,A -85,B 0,C 180,E1 -21076.578,E2 -21076.578} C_VEL
LIN {X 0,Y 232.82,Z 217.03,A -85,B 0,C 180,E1 -21078.524,E2 -21078.524} C_VEL
LIN {X 0,Y 238.254,Z 228.51,A -85,B 0,C 180,E1 -21080.479,E2 -21080.479} C_VEL
LIN {X 0,Y 239.585,Z 231.842,A -85,B 0,C 180,E1 -21080.96,E2 -21080.96} C_VEL
LIN {X 0,Y 236.094,Z 284.736,A -85,B 0,C 180,E1 -21082.659,E2 -21082.659} C_VEL
LIN {X 0,Y 234.481,Z 297.786,A -85,B 0,C 180,E1 -21083.376,E2 -21083.376} C_VEL
LIN {X 0,Y 232.446,Z 310.014,A -85,B 0,C 180,E1 -21084.378,E2 -21084.378} C_VEL
LIN {X 0,Y 229.835,Z 321.869,A -85,B 0,C 180,E1 -21085.698,E2 -21085.698} C_VEL
LIN {X 0,Y 226.776,Z 333.121,A -85,B 0,C 180,E1 -21087.325,E2 -21087.325} C_VEL
LIN {X 0,Y 223.529,Z 343.279,A -85,B 0,C 180,E1 -21089.194,E2 -21089.194} C_VEL
LIN {X 0,Y 220.184,Z 352.544,A -85,B 0,C 180,E1 -21091.369,E2 -21091.369} C_VEL
LIN {X 0,Y 216.512,Z 361.734,A -85,B 0,C 180,E1 -21094.133,E2 -21094.133} C_VEL
LIN {X 0,Y 213.435,Z 368.834,A -85,B 0,C 180,E1 -21096.879,E2 -21096.879} C_VEL
LIN {X 0,Y 210.637,Z 374.809,A -85,B 0,C 180,E1 -21099.878,E2 -21099.878} C_VEL
LIN {X 0,Y 208.08,Z 380.077,A -85,B 0,C 180,E1 -21103.463,E2 -21103.463} C_VEL
LIN {X 0,Y 206.235,Z 383.649,A -85,B 0,C 180,E1 -21107.034,E2 -21107.034} C_VEL
LIN {X 0,Y 205.328,Z 385.203,A -85,B 0,C 180,E1 -21109.433,E2 -21109.433} C_VEL
LIN {X 0,Y 204.566,Z 386.252,A -85,B 0,C 180,E1 -21112.203,E2 -21112.203} C_VEL
LIN {X 0,Y 204.042,Z 386.45,A -85,B 0,C 180,E1 -21115.757,E2 -21115.757} C_VEL
LIN {X 0,Y 203.971,Z 385.297,A -85,B 0,C 180,E1 -21119.474,E2 -21119.474} C_VEL
LIN {X 0,Y 204.102,Z 384.273,A -85,B 0,C 180,E1 -21121.179,E2 -21121.179} C_VEL
LIN {X 0,Y 204.685,Z 381.264,A -85,B 0,C 180,E1 -21124.583,E2 -21124.583} C_VEL
LIN {X 0,Y 205.482,Z 377.017,A -85,B 0,C 180,E1 -21127.9,E2 -21127.9} C_VEL
LIN {X 0,Y 206.564,Z 371.524,A -85,B 0,C 180,E1 -21131.1,E2 -21131.1} C_VEL
LIN {X 0,Y 207.91,Z 365.578,A -85,B 0,C 180,E1 -21133.807,E2 -21133.807} C_VEL
LIN {X 0,Y 209.638,Z 358.321,A -85,B 0,C 180,E1 -21136.462,E2 -21136.462} C_VEL
LIN {X 0,Y 211.592,Z 349.7,A -85,B 0,C 180,E1 -21138.99,E2 -21138.99} C_VEL
LIN {X 0,Y 213.836,Z 339.387,A -85,B 0,C 180,E1 -21141.401,E2 -21141.401} C_VEL
LIN {X 0,Y 215.78,Z 329.638,A -85,B 0,C 180,E1 -21143.219,E2 -21143.219} C_VEL
LIN {X 0,Y 217.771,Z 318.102,A -85,B 0,C 180,E1 -21144.918,E2 -21144.918} C_VEL
LIN {X 0,Y 219.548,Z 305.482,A -85,B 0,C 180,E1 -21146.329,E2 -21146.329} C_VEL
LIN {X 0,Y 220.987,Z 292.747,A -85,B 0,C 180,E1 -21147.351,E2 -21147.351} C_VEL
LIN {X 0,Y 221.96,Z 279.96,A -85,B 0,C 180,E1 -21148.015,E2 -21148.015} C_VEL
LIN {X 0,Y 224.583,Z 219.482,A -85,B 0,C 180,E1 -21150.041,E2 -21150.041} C_VEL
LIN {X 0,Y 215.068,Z 193.766,A -85,B 0,C 180,E1 -21152.344,E2 -21152.344} C_VEL
LIN {X 0,Y 210.729,Z 184.975,A -85,B 0,C 180,E1 -21153.348,E2 -21153.348} C_VEL
LIN {X 0,Y 207.33,Z 178.962,A -85,B 0,C 180,E1 -21154.131,E2 -21154.131} C_VEL
LIN {X 0,Y 207.038,Z 177.695,A -85,B 0,C 180,E1 -21154.258,E2 -21154.258} C_VEL
LIN {X 0,Y 207.131,Z 177.684,A -85,B 0,C 180,E1 -21157.8,E2 -21157.8} C_VEL
LIN {X 0,Y 206.912,Z 177.703,A -85,B 0,C 180,E1 -21161.759,E2 -21161.759} C_VEL
LIN {X 0,Y 206.814,Z 177.715,A -85,B 0,C 180,E1 -21165.775,E2 -21165.775} C_VEL
LIN {X 0,Y 206.746,Z 177.734,A -85,B 0,C 180,E1 -21169.873,E2 -21169.873} C_VEL
LIN {X 0,Y 206.693,Z 177.723,A -85,B 0,C 180,E1 -21174.081,E2 -21174.081} C_VEL
LIN {X 0,Y 206.688,Z 177.738,A -85,B 0,C 180,E1 -21178.427,E2 -21178.427} C_VEL
LIN {X 0,Y 206.697,Z 177.716,A -85,B 0,C 180,E1 -21182.958,E2 -21182.958} C_VEL
LIN {X 0,Y 206.675,Z 177.739,A -85,B 0,C 180,E1 -21187.741,E2 -21187.741} C_VEL
LIN {X 0,Y 206.633,Z 177.741,A -85,B 0,C 180,E1 -21191.559,E2 -21191.559} C_VEL
LIN {X 0,Y 206.631,Z 177.712,A -85,B 0,C 180,E1 -21195.583,E2 -21195.583} C_VEL
LIN {X 0,Y 206.648,Z 177.731,A -85,B 0,C 180,E1 -21199.746,E2 -21199.746} C_VEL
LIN {X 0,Y 206.701,Z 177.738,A -85,B 0,C 180,E1 -21204.689,E2 -21204.689} C_VEL
LIN {X 0,Y 206.698,Z 177.732,A -85,B 0,C 180,E1 -21209.335,E2 -21209.335} C_VEL
LIN {X 0,Y 206.707,Z 177.734,A -85,B 0,C 180,E1 -21213.768,E2 -21213.768} C_VEL
LIN {X 0,Y 206.718,Z 177.727,A -85,B 0,C 180,E1 -21218.039,E2 -21218.039} C_VEL
LIN {X 0,Y 206.805,Z 177.724,A -85,B 0,C 180,E1 -21222.19,E2 -21222.19} C_VEL
LIN {X 0,Y 206.86,Z 177.707,A -85,B 0,C 180,E1 -21226.242,E2 -21226.242} C_VEL
LIN {X 0,Y 207.082,Z 177.691,A -85,B 0,C 180,E1 -21230.23,E2 -21230.23} C_VEL
LIN {X 0,Y 207.042,Z 177.685,A -85,B 0,C 180,E1 -21234.155,E2 -21234.155} C_VEL
LIN {X 0,Y 207.347,Z 177.657,A -85,B 0,C 180,E1 -21238.058,E2 -21238.058} C_VEL
LIN {X 0,Y 207.483,Z 177.64,A -85,B 0,C 180,E1 -21240,E2 -21240} C_VEL
LIN {X 0,Y 207.346,Z 177.648,A -85,B 0,C 180,E1 -21241.942,E2 -21241.942} C_VEL
LIN {X 0,Y 207.125,Z 177.651,A -85,B 0,C 180,E1 -21247.8,E2 -21247.8} C_VEL
LIN {X 0,Y 206.899,Z 177.708,A -85,B 0,C 180,E1 -21251.76,E2 -21251.76} C_VEL
LIN {X 0,Y 206.805,Z 177.722,A -85,B 0,C 180,E1 -21255.776,E2 -21255.776} C_VEL
LIN {X 0,Y 206.711,Z 177.709,A -85,B 0,C 180,E1 -21259.876,E2 -21259.876} C_VEL
LIN {X 0,Y 206.722,Z 177.732,A -85,B 0,C 180,E1 -21264.077,E2 -21264.077} C_VEL
LIN {X 0,Y 206.687,Z 177.733,A -85,B 0,C 180,E1 -21268.427,E2 -21268.427} C_VEL
LIN {X 0,Y 206.696,Z 177.738,A -85,B 0,C 180,E1 -21272.958,E2 -21272.958} C_VEL
LIN {X 0,Y 206.669,Z 177.743,A -85,B 0,C 180,E1 -21277.742,E2 -21277.742} C_VEL
LIN {X 0,Y 206.632,Z 177.744,A -85,B 0,C 180,E1 -21281.559,E2 -21281.559} C_VEL
LIN {X 0,Y 206.63,Z 177.736,A -85,B 0,C 180,E1 -21285.583,E2 -21285.583} C_VEL
LIN {X 0,Y 206.721,Z 177.8,A -85,B 0,C 180,E1 -21290.139,E2 -21290.139} C_VEL
LIN {X 0,Y 208.512,Z 185.456,A -85,B 0,C 180,E1 -21293.911,E2 -21293.911} C_VEL
LIN {X 0,Y 210.486,Z 190.26,A -85,B 0,C 180,E1 -21294.433,E2 -21294.433} C_VEL
LIN {X 0,Y 212.255,Z 195.586,A -85,B 0,C 180,E1 -21294.92,E2 -21294.92} C_VEL
LIN {X 0,Y 213.618,Z 205.111,A -85,B 0,C 180,E1 -21295.513,E2 -21295.513} C_VEL
LIN {X 0,Y 214.158,Z 212.974,A -85,B 0,C 180,E1 -21295.914,E2 -21295.914} C_VEL
LIN {X 0,Y 215.102,Z 220.744,A -85,B 0,C 180,E1 -21296.362,E2 -21296.362} C_VEL
LIN {X 0,Y 217.538,Z 240.33,A -85,B 0,C 180,E1 -21297.472,E2 -21297.472} C_VEL
LIN {X 0,Y 215.037,Z 294.237,A -85,B 0,C 180,E1 -21299.359,E2 -21299.359} C_VEL
LIN {X 0,Y 213.753,Z 307.717,A -85,B 0,C 180,E1 -21300.178,E2 -21300.178} C_VEL
LIN {X 0,Y 212.113,Z 320.075,A -85,B 0,C 180,E1 -21301.286,E2 -21301.286} C_VEL
LIN {X 0,Y 210.254,Z 331.197,A -85,B 0,C 180,E1 -21302.638,E2 -21302.638} C_VEL
LIN {X 0,Y 207.809,Z 342.781,A -85,B 0,C 180,E1 -21304.456,E2 -21304.456} C_VEL
LIN {X 0,Y 205.617,Z 353.294,A -85,B 0,C 180,E1 -21306.588,E2 -21306.588} C_VEL
LIN {X 0,Y 203.709,Z 361.571,A -85,B 0,C 180,E1 -21308.671,E2 -21308.671} C_VEL
LIN {X 0,Y 201.854,Z 369.787,A -85,B 0,C 180,E1 -21311.212,E2 -21311.212} C_VEL
LIN {X 0,Y 200.024,Z 377.476,A -85,B 0,C 180,E1 -21314.199,E2 -21314.199} C_VEL
LIN {X 0,Y 198.508,Z 384.564,A -85,B 0,C 180,E1 -21317.735,E2 -21317.735} C_VEL
LIN {X 0,Y 197.773,Z 389.234,A -85,B 0,C 180,E1 -21320.798,E2 -21320.798} C_VEL
LIN {X 0,Y 197.366,Z 392.755,A -85,B 0,C 180,E1 -21323.868,E2 -21323.868} C_VEL
LIN {X 0,Y 197.249,Z 394.617,A -85,B 0,C 180,E1 -21326.068,E2 -21326.068} C_VEL
LIN {X 0,Y 197.399,Z 396.741,A -85,B 0,C 180,E1 -21330,E2 -21330} C_VEL
LIN {X 0,Y 197.261,Z 397.239,A -85,B 0,C 180,E1 -21332.042,E2 -21332.042} C_VEL
LIN {X 0,Y 197.249,Z 397.302,A -85,B 0,C 180,E1 -21334.086,E2 -21334.086} C_VEL
LIN {X 0,Y 197.594,Z 396.261,A -85,B 0,C 180,E1 -21338.179,E2 -21338.179} C_VEL
LIN {X 0,Y 198.052,Z 395.164,A -85,B 0,C 180,E1 -21340.22,E2 -21340.22} C_VEL
LIN {X 0,Y 198.717,Z 393.627,A -85,B 0,C 180,E1 -21342.252,E2 -21342.252} C_VEL
LIN {X 0,Y 200.067,Z 390.546,A -85,B 0,C 180,E1 -21345.276,E2 -21345.276} C_VEL
LIN {X 0,Y 202.103,Z 386.441,A -85,B 0,C 180,E1 -21348.238,E2 -21348.238} C_VEL
LIN {X 0,Y 205.081,Z 380.193,A -85,B 0,C 180,E1 -21351.617,E2 -21351.617} C_VEL
LIN {X 0,Y 208.051,Z 373.441,A -85,B 0,C 180,E1 -21354.444,E2 -21354.444} C_VEL
LIN {X 0,Y 211.648,Z 365.099,A -85,B 0,C 180,E1 -21357.167,E2 -21357.167} C_VEL
LIN {X 0,Y 215.115,Z 356.546,A -85,B 0,C 180,E1 -21359.345,E2 -21359.345} C_VEL
LIN {X 0,Y 218.829,Z 346.077,A -85,B 0,C 180,E1 -21361.46,E2 -21361.46} C_VEL
LIN {X 0,Y 222.554,Z 334.33,A -85,B 0,C 180,E1 -21363.277,E2 -21363.277} C_VEL
LIN {X 0,Y 225.547,Z 322.656,A -85,B 0,C 180,E1 -21364.658,E2 -21364.658} C_VEL
LIN {X 0,Y 228.042,Z 310.701,A -85,B 0,C 180,E1 -21365.707,E2 -21365.707} C_VEL
LIN {X 0,Y 230.086,Z 297.924,A -85,B 0,C 180,E1 -21366.485,E2 -21366.485} C_VEL
LIN {X 0,Y 231.323,Z 283.65,A -85,B 0,C 180,E1 -21367.05,E2 -21367.05} C_VEL
LIN {X 0,Y 233.8,Z 244.513,A -85,B 0,C 180,E1 -21368.32,E2 -21368.32} C_VEL
LIN {X 0,Y 233.11,Z 238.776,A -85,B 0,C 180,E1 -21368.777,E2 -21368.777} C_VEL
LIN {X 0,Y 229.508,Z 229.644,A -85,B 0,C 180,E1 -21370.198,E2 -21370.198} C_VEL
LIN {X 0,Y 224.535,Z 218.996,A -85,B 0,C 180,E1 -21372.254,E2 -21372.254} C_VEL
LIN {X 0,Y 219.344,Z 209.548,A -85,B 0,C 180,E1 -21374.533,E2 -21374.533} C_VEL
LIN {X 0,Y 216.172,Z 204.419,A -85,B 0,C 180,E1 -21376.035,E2 -21376.035} C_VEL
LIN {X 0,Y 213.173,Z 199.685,A -85,B 0,C 180,E1 -21377.549,E2 -21377.549} C_VEL
LIN {X 0,Y 209.406,Z 194.054,A -85,B 0,C 180,E1 -21379.654,E2 -21379.654} C_VEL
LIN {X 0,Y 206.109,Z 189.225,A -85,B 0,C 180,E1 -21381.702,E2 -21381.702} C_VEL
LIN {X 0,Y 201.465,Z 183.371,A -85,B 0,C 180,E1 -21384.972,E2 -21384.972} C_VEL
LIN {X 0,Y 200.804,Z 181.939,A -85,B 0,C 180,E1 -21385.725,E2 -21385.725} C_VEL
LIN {X 0,Y 199.624,Z 178.606,A -85,B 0,C 180,E1 -21390.179,E2 -21390.179} C_VEL
LIN {X 0,Y 199.622,Z 178.603,A -85,B 0,C 180,E1 -21395.009,E2 -21395.009} C_VEL
LIN {X 0,Y 199.643,Z 178.6,A -85,B 0,C 180,E1 -21399.389,E2 -21399.389} C_VEL
LIN {X 0,Y 199.741,Z 178.589,A -85,B 0,C 180,E1 -21403.651,E2 -21403.651} C_VEL
LIN {X 0,Y 200.025,Z 178.554,A -85,B 0,C 180,E1 -21409.882,E2 -21409.882} C_VEL
LIN {X 0,Y 200.004,Z 178.553,A -85,B 0,C 180,E1 -21413.949,E2 -21413.949} C_VEL
LIN {X 0,Y 200.287,Z 178.519,A -85,B 0,C 180,E1 -21417.989,E2 -21417.989} C_VEL
LIN {X 0,Y 200.45,Z 178.515,A -85,B 0,C 180,E1 -21420,E2 -21420} C_VEL
LIN {X 0,Y 200.256,Z 178.547,A -85,B 0,C 180,E1 -21422.137,E2 -21422.137} C_VEL
LIN {X 0,Y 200.861,Z 180.919,A -85,B 0,C 180,E1 -21422.82,E2 -21422.82} C_VEL
LIN {X 0,Y 202.468,Z 183.112,A -85,B 0,C 180,E1 -21424.118,E2 -21424.118} C_VEL
LIN {X 0,Y 204.69,Z 184.584,A -85,B 0,C 180,E1 -21425.585,E2 -21425.585} C_VEL
LIN {X 0,Y 206.222,Z 187.347,A -85,B 0,C 180,E1 -21426.666,E2 -21426.666} C_VEL
LIN {X 0,Y 208.956,Z 190.03,A -85,B 0,C 180,E1 -21428.279,E2 -21428.279} C_VEL
LIN {X 0,Y 211.174,Z 193.433,A -85,B 0,C 180,E1 -21429.579,E2 -21429.579} C_VEL
LIN {X 0,Y 212.739,Z 195.322,A -85,B 0,C 180,E1 -21430.414,E2 -21430.414} C_VEL
LIN {X 0,Y 216.701,Z 200.82,A -85,B 0,C 180,E1 -21432.394,E2 -21432.394} C_VEL
LIN {X 0,Y 220.826,Z 207.341,A -85,B 0,C 180,E1 -21434.315,E2 -21434.315} C_VEL
LIN {X 0,Y 226.061,Z 216.25,A -85,B 0,C 180,E1 -21436.524,E2 -21436.524} C_VEL
LIN {X 0,Y 231.461,Z 227.27,A -85,B 0,C 180,E1 -21438.674,E2 -21438.674} C_VEL
LIN {X 0,Y 234.465,Z 234.227,A -85,B 0,C 180,E1 -21439.807,E2 -21439.807} C_VEL
LIN {X 0,Y 230.956,Z 284.926,A -85,B 0,C 180,E1 -21441.458,E2 -21441.458} C_VEL
LIN {X 0,Y 229.161,Z 298.764,A -85,B 0,C 180,E1 -21442.24,E2 -21442.24} C_VEL
LIN {X 0,Y 226.876,Z 311.486,A -85,B 0,C 180,E1 -21443.336,E2 -21443.336} C_VEL
LIN {X 0,Y 224.22,Z 322.743,A -85,B 0,C 180,E1 -21444.634,E2 -21444.634} C_VEL
LIN {X 0,Y 220.764,Z 334.608,A -85,B 0,C 180,E1 -21446.406,E2 -21446.406} C_VEL
LIN {X 0,Y 217.473,Z 344.329,A -85,B 0,C 180,E1 -21448.281,E2 -21448.281} C_VEL
LIN {X 0,Y 213.607,Z 354.295,A -85,B 0,C 180,E1 -21450.733,E2 -21450.733} C_VEL
LIN {X 0,Y 210.183,Z 362.393,A -85,B 0,C 180,E1 -21453.285,E2 -21453.285} C_VEL
LIN {X 0,Y 206.848,Z 369.593,A -85,B 0,C 180,E1 -21456.201,E2 -21456.201} C_VEL
LIN {X 0,Y 203.951,Z 375.374,A -85,B 0,C 180,E1 -21459.248,E2 -21459.248} C_VEL
LIN {X 0,Y 201.295,Z 380.424,A -85,B 0,C 180,E1 -21462.845,E2 -21462.845} C_VEL
LIN {X 0,Y 199.904,Z 382.932,A -85,B 0,C 180,E1 -21465.32,E2 -21465.32} C_VEL
LIN {X 0,Y 198.748,Z 384.9,A -85,B 0,C 180,E1 -21467.953,E2 -21467.953} C_VEL
LIN {X 0,Y 197.631,Z 386.392,A -85,B 0,C 180,E1 -21471.476,E2 -21471.476} C_VEL
LIN {X 0,Y 196.984,Z 386.676,A -85,B 0,C 180,E1 -21475.19,E2 -21475.19} C_VEL
LIN {X 0,Y 196.847,Z 385.638,A -85,B 0,C 180,E1 -21478.967,E2 -21478.967} C_VEL
LIN {X 0,Y 197.271,Z 383.011,A -85,B 0,C 180,E1 -21482.956,E2 -21482.956} C_VEL
LIN {X 0,Y 197.893,Z 380.022,A -85,B 0,C 180,E1 -21485.895,E2 -21485.895} C_VEL
LIN {X 0,Y 198.782,Z 375.28,A -85,B 0,C 180,E1 -21489.295,E2 -21489.295} C_VEL
LIN {X 0,Y 200.218,Z 368.835,A -85,B 0,C 180,E1 -21492.774,E2 -21492.774} C_VEL
LIN {X 0,Y 202.045,Z 361.262,A -85,B 0,C 180,E1 -21495.907,E2 -21495.907} C_VEL
LIN {X 0,Y 203.99,Z 353.131,A -85,B 0,C 180,E1 -21498.574,E2 -21498.574} C_VEL
LIN {X 0,Y 206.262,Z 343.262,A -85,B 0,C 180,E1 -21501.163,E2 -21501.163} C_VEL
LIN {X 0,Y 208.435,Z 333.313,A -85,B 0,C 180,E1 -21503.222,E2 -21503.222} C_VEL
LIN {X 0,Y 210.576,Z 321.814,A -85,B 0,C 180,E1 -21505.104,E2 -21505.104} C_VEL
LIN {X 0,Y 212.517,Z 309.269,A -85,B 0,C 180,E1 -21506.682,E2 -21506.682} C_VEL
LIN {X 0,Y 214.143,Z 295.879,A -85,B 0,C 180,E1 -21507.884,E2 -21507.884} C_VEL
LIN {X 0,Y 215.312,Z 283.126,A -85,B 0,C 180,E1 -21508.649,E2 -21508.649} C_VEL
LIN {X 0,Y 218.246,Z 221.153,A -85,B 0,C 180,E1 -21510.796,E2 -21510.796} C_VEL
LIN {X 0,Y 208.487,Z 194.975,A -85,B 0,C 180,E1 -21513.262,E2 -21513.262} C_VEL
LIN {X 0,Y 203.029,Z 185.08,A -85,B 0,C 180,E1 -21514.545,E2 -21514.545} C_VEL
LIN {X 0,Y 200.124,Z 179.291,A -85,B 0,C 180,E1 -21515.283,E2 -21515.283} C_VEL
LIN {X 0,Y 200,Z 178.576,A -85,B 0,C 180,E1 -21515.345,E2 -21515.345} C_VEL
LIN {X 0,Y 200.079,Z 178.564,A -85,B 0,C 180,E1 -21518.077,E2 -21518.077} C_VEL
LIN {X 0,Y 199.86,Z 178.583,A -85,B 0,C 180,E1 -21522.18,E2 -21522.18} C_VEL
LIN {X 0,Y 199.756,Z 178.589,A -85,B 0,C 180,E1 -21526.348,E2 -21526.348} C_VEL
LIN {X 0,Y 199.665,Z 178.614,A -85,B 0,C 180,E1 -21530.609,E2 -21530.609} C_VEL
LIN {X 0,Y 199.623,Z 178.606,A -85,B 0,C 180,E1 -21534.991,E2 -21534.991} C_VEL
LIN {X 0,Y 199.609,Z 178.62,A -85,B 0,C 180,E1 -21539.533,E2 -21539.533} C_VEL
LIN {X 0,Y 199.667,Z 178.595,A -85,B 0,C 180,E1 -21542.353,E2 -21542.353} C_VEL
LIN {X 0,Y 199.622,Z 178.612,A -85,B 0,C 180,E1 -21546.764,E2 -21546.764} C_VEL
LIN {X 0,Y 199.598,Z 178.624,A -85,B 0,C 180,E1 -21549.331,E2 -21549.331} C_VEL
LIN {X 0,Y 199.568,Z 178.618,A -85,B 0,C 180,E1 -21552.308,E2 -21552.308} C_VEL
LIN {X 0,Y 199.577,Z 178.591,A -85,B 0,C 180,E1 -21555.227,E2 -21555.227} C_VEL
LIN {X 0,Y 199.571,Z 178.597,A -85,B 0,C 180,E1 -21558.002,E2 -21558.002} C_VEL
LIN {X 0,Y 199.598,Z 178.613,A -85,B 0,C 180,E1 -21560.773,E2 -21560.773} C_VEL
LIN {X 0,Y 199.612,Z 178.616,A -85,B 0,C 180,E1 -21565.713,E2 -21565.713} C_VEL
LIN {X 0,Y 199.688,Z 178.598,A -85,B 0,C 180,E1 -21568.134,E2 -21568.134} C_VEL
LIN {X 0,Y 199.646,Z 178.618,A -85,B 0,C 180,E1 -21572.765,E2 -21572.765} C_VEL
LIN {X 0,Y 199.68,Z 178.602,A -85,B 0,C 180,E1 -21577.222,E2 -21577.222} C_VEL
LIN {X 0,Y 199.747,Z 178.602,A -85,B 0,C 180,E1 -21581.803,E2 -21581.803} C_VEL
LIN {X 0,Y 199.777,Z 178.587,A -85,B 0,C 180,E1 -21585.744,E2 -21585.744} C_VEL
LIN {X 0,Y 200.025,Z 178.568,A -85,B 0,C 180,E1 -21589.882,E2 -21589.882} C_VEL
LIN {X 0,Y 200.006,Z 178.561,A -85,B 0,C 180,E1 -21593.949,E2 -21593.949} C_VEL
LIN {X 0,Y 200.289,Z 178.536,A -85,B 0,C 180,E1 -21597.989,E2 -21597.989} C_VEL
LIN {X 0,Y 200.45,Z 178.515,A -85,B 0,C 180,E1 -21600,E2 -21600} C_VEL
LIN {X 0,Y 199.99,Z 178.548,A -85,B 0,C 180,E1 -21604.03,E2 -21604.03} C_VEL
LIN {X 0,Y 200.073,Z 178.53,A -85,B 0,C 180,E1 -21608.077,E2 -21608.077} C_VEL
LIN {X 0,Y 199.85,Z 178.589,A -85,B 0,C 180,E1 -21612.181,E2 -21612.181} C_VEL
LIN {X 0,Y 199.744,Z 178.598,A -85,B 0,C 180,E1 -21616.349,E2 -21616.349} C_VEL
LIN {X 0,Y 199.644,Z 178.588,A -85,B 0,C 180,E1 -21620.611,E2 -21620.611} C_VEL
LIN {X 0,Y 199.636,Z 178.615,A -85,B 0,C 180,E1 -21624.989,E2 -21624.989} C_VEL
LIN {X 0,Y 199.608,Z 178.617,A -85,B 0,C 180,E1 -21629.533,E2 -21629.533} C_VEL
LIN {X 0,Y 199.667,Z 178.614,A -85,B 0,C 180,E1 -21632.352,E2 -21632.352} C_VEL
LIN {X 0,Y 199.619,Z 178.622,A -85,B 0,C 180,E1 -21636.764,E2 -21636.764} C_VEL
LIN {X 0,Y 199.595,Z 178.624,A -85,B 0,C 180,E1 -21639.331,E2 -21639.331} C_VEL
LIN {X 0,Y 199.567,Z 178.625,A -85,B 0,C 180,E1 -21642.307,E2 -21642.307} C_VEL
LIN {X 0,Y 199.576,Z 178.614,A -85,B 0,C 180,E1 -21645.227,E2 -21645.227} C_VEL
LIN {X 0,Y 199.641,Z 178.713,A -85,B 0,C 180,E1 -21649.364,E2 -21649.364} C_VEL
LIN {X 0,Y 201.321,Z 185.555,A -85,B 0,C 180,E1 -21652.785,E2 -21652.785} C_VEL
LIN {X 0,Y 208.937,Z 203.631,A -85,B 0,C 180,E1 -21654.771,E2 -21654.771} C_VEL
LIN {X 0,Y 214.964,Z 220.005,A -85,B 0,C 180,E1 -21656.313,E2 -21656.313} C_VEL
LIN {X 0,Y 215.102,Z 220.744,A -85,B 0,C 180,E1 -21656.362,E2 -21656.362} C_VEL
LIN {X 0,Y 215.409,Z 226.547,A -85,B 0,C 180,E1 -21656.64,E2 -21656.64} C_VEL
LIN {X 0,Y 214.613,Z 232.432,A -85,B 0,C 180,E1 -21656.772,E2 -21656.772} C_VEL
LIN {X 0,Y 211.023,Z 248.185,A -85,B 0,C 180,E1 -21656.937,E2 -21656.937} C_VEL
LIN {X 0,Y 210.631,Z 252.186,A -85,B 0,C 180,E1 -21657.05,E2 -21657.05} C_VEL
LIN {X 0,Y 208.569,Z 294.371,A -85,B 0,C 180,E1 -21658.584,E2 -21658.584} C_VEL
LIN {X 0,Y 207.129,Z 308.473,A -85,B 0,C 180,E1 -21659.476,E2 -21659.476} C_VEL
LIN {X 0,Y 205.542,Z 320.034,A -85,B 0,C 180,E1 -21660.559,E2 -21660.559} C_VEL
LIN {X 0,Y 203.267,Z 332.689,A -85,B 0,C 180,E1 -21662.175,E2 -21662.175} C_VEL
LIN {X 0,Y 200.87,Z 343.993,A -85,B 0,C 180,E1 -21664.065,E2 -21664.065} C_VEL
LIN {X 0,Y 198.608,Z 354.214,A -85,B 0,C 180,E1 -21666.264,E2 -21666.264} C_VEL
LIN {X 0,Y 196.154,Z 364.243,A -85,B 0,C 180,E1 -21669.005,E2 -21669.005} C_VEL
LIN {X 0,Y 194.349,Z 371.705,A -85,B 0,C 180,E1 -21671.554,E2 -21671.554} C_VEL
LIN {X 0,Y 192.575,Z 379.022,A -85,B 0,C 180,E1 -21674.657,E2 -21674.657} C_VEL
LIN {X 0,Y 191.545,Z 383.947,A -85,B 0,C 180,E1 -21677.282,E2 -21677.282} C_VEL
LIN {X 0,Y 190.731,Z 388.71,A -85,B 0,C 180,E1 -21680.455,E2 -21680.455} C_VEL
LIN {X 0,Y 190.297,Z 392.315,A -85,B 0,C 180,E1 -21683.639,E2 -21683.639} C_VEL
LIN {X 0,Y 190.161,Z 394.488,A -85,B 0,C 180,E1 -21686.263,E2 -21686.263} C_VEL
LIN {X 0,Y 190.299,Z 396.453,A -85,B 0,C 180,E1 -21690,E2 -21690} C_VEL
LIN {X 0,Y 190.135,Z 397.113,A -85,B 0,C 180,E1 -21693.618,E2 -21693.618} C_VEL
LIN {X 0,Y 190.279,Z 396.83,A -85,B 0,C 180,E1 -21696.362,E2 -21696.362} C_VEL
LIN {X 0,Y 191.047,Z 395.097,A -85,B 0,C 180,E1 -21700.599,E2 -21700.599} C_VEL
LIN {X 0,Y 191.751,Z 393.639,A -85,B 0,C 180,E1 -21702.704,E2 -21702.704} C_VEL
LIN {X 0,Y 193.215,Z 390.64,A -85,B 0,C 180,E1 -21705.831,E2 -21705.831} C_VEL
LIN {X 0,Y 195.373,Z 386.621,A -85,B 0,C 180,E1 -21708.89,E2 -21708.89} C_VEL
LIN {X 0,Y 198.471,Z 380.495,A -85,B 0,C 180,E1 -21712.375,E2 -21712.375} C_VEL
LIN {X 0,Y 201.618,Z 373.849,A -85,B 0,C 180,E1 -21715.278,E2 -21715.278} C_VEL
LIN {X 0,Y 205.374,Z 365.641,A -85,B 0,C 180,E1 -21718.069,E2 -21718.069} C_VEL
LIN {X 0,Y 209.011,Z 357.302,A -85,B 0,C 180,E1 -21720.29,E2 -21720.29} C_VEL
LIN {X 0,Y 212.863,Z 347.106,A -85,B 0,C 180,E1 -21722.447,E2 -21722.447} C_VEL
LIN {X 0,Y 216.73,Z 335.675,A -85,B 0,C 180,E1 -21724.293,E2 -21724.293} C_VEL
LIN {X 0,Y 219.843,Z 324.516,A -85,B 0,C 180,E1 -21725.692,E2 -21725.692} C_VEL
LIN {X 0,Y 222.647,Z 311.974,A -85,B 0,C 180,E1 -21726.852,E2 -21726.852} C_VEL
LIN {X 0,Y 224.921,Z 298.519,A -85,B 0,C 180,E1 -21727.709,E2 -21727.709} C_VEL
LIN {X 0,Y 226.238,Z 284.935,A -85,B 0,C 180,E1 -21728.27,E2 -21728.27} C_VEL
LIN {X 0,Y 228.845,Z 245.365,A -85,B 0,C 180,E1 -21729.575,E2 -21729.575} C_VEL
LIN {X 0,Y 228.305,Z 241.618,A -85,B 0,C 180,E1 -21729.914,E2 -21729.914} C_VEL
LIN {X 0,Y 225.176,Z 233.465,A -85,B 0,C 180,E1 -21731.258,E2 -21731.258} C_VEL
LIN {X 0,Y 220.667,Z 223.631,A -85,B 0,C 180,E1 -21733.232,E2 -21733.232} C_VEL
LIN {X 0,Y 216.106,Z 214.986,A -85,B 0,C 180,E1 -21735.382,E2 -21735.382} C_VEL
LIN {X 0,Y 212.912,Z 209.712,A -85,B 0,C 180,E1 -21736.976,E2 -21736.976} C_VEL
LIN {X 0,Y 210.349,Z 205.458,A -85,B 0,C 180,E1 -21738.37,E2 -21738.37} C_VEL
LIN {X 0,Y 206.75,Z 199.965,A -85,B 0,C 180,E1 -21740.485,E2 -21740.485} C_VEL
LIN {X 0,Y 203.273,Z 194.827,A -85,B 0,C 180,E1 -21742.777,E2 -21742.777} C_VEL
LIN {X 0,Y 199.385,Z 189.619,A -85,B 0,C 180,E1 -21745.744,E2 -21745.744} C_VEL
LIN {X 0,Y 198.496,Z 188.163,A -85,B 0,C 180,E1 -21746.543,E2 -21746.543} C_VEL
LIN {X 0,Y 195.001,Z 184.174,A -85,B 0,C 180,E1 -21749.881,E2 -21749.881} C_VEL
LIN {X 0,Y 193.084,Z 181.341,A -85,B 0,C 180,E1 -21752.349,E2 -21752.349} C_VEL
LIN {X 0,Y 192.639,Z 179.478,A -85,B 0,C 180,E1 -21756.34,E2 -21756.34} C_VEL
LIN {X 0,Y 192.696,Z 179.478,A -85,B 0,C 180,E1 -21761.492,E2 -21761.492} C_VEL
LIN {X 0,Y 192.775,Z 179.463,A -85,B 0,C 180,E1 -21767.365,E2 -21767.365} C_VEL
LIN {X 0,Y 193.027,Z 179.434,A -85,B 0,C 180,E1 -21771.626,E2 -21771.626} C_VEL
LIN {X 0,Y 192.971,Z 179.581,A -85,B 0,C 180,E1 -21775.692,E2 -21775.692} C_VEL
LIN {X 0,Y 193.696,Z 181.635,A -85,B 0,C 180,E1 -21776.88,E2 -21776.88} C_VEL
LIN {X 0,Y 196.307,Z 184.279,A -85,B 0,C 180,E1 -21779.744,E2 -21779.744} C_VEL
LIN {X 0,Y 198.191,Z 185.536,A -85,B 0,C 180,E1 -21781.396,E2 -21781.396} C_VEL
LIN {X 0,Y 199.551,Z 188.472,A -85,B 0,C 180,E1 -21782.713,E2 -21782.713} C_VEL
LIN {X 0,Y 201.92,Z 190.667,A -85,B 0,C 180,E1 -21784.492,E2 -21784.492} C_VEL
LIN {X 0,Y 202.69,Z 191.504,A -85,B 0,C 180,E1 -21785.035,E2 -21785.035} C_VEL
LIN {X 0,Y 205.086,Z 194.923,A -85,B 0,C 180,E1 -21786.703,E2 -21786.703} C_VEL
LIN {X 0,Y 206.621,Z 196.518,A -85,B 0,C 180,E1 -21787.635,E2 -21787.635} C_VEL
LIN {X 0,Y 209.269,Z 200.262,A -85,B 0,C 180,E1 -21789.21,E2 -21789.21} C_VEL
LIN {X 0,Y 213.87,Z 206.776,A -85,B 0,C 180,E1 -21791.675,E2 -21791.675} C_VEL
LIN {X 0,Y 216.869,Z 211.606,A -85,B 0,C 180,E1 -21793.148,E2 -21793.148} C_VEL
LIN {X 0,Y 222.312,Z 221.172,A -85,B 0,C 180,E1 -21795.623,E2 -21795.623} C_VEL
LIN {X 0,Y 227.319,Z 231.638,A -85,B 0,C 180,E1 -21797.735,E2 -21797.735} C_VEL
LIN {X 0,Y 229.396,Z 236.514,A -85,B 0,C 180,E1 -21798.585,E2 -21798.585} C_VEL
LIN {X 0,Y 225.906,Z 285.34,A -85,B 0,C 180,E1 -21800.211,E2 -21800.211} C_VEL
LIN {X 0,Y 224.068,Z 298.995,A -85,B 0,C 180,E1 -21800.995,E2 -21800.995} C_VEL
LIN {X 0,Y 221.79,Z 311.231,A -85,B 0,C 180,E1 -21802.05,E2 -21802.05} C_VEL
LIN {X 0,Y 219.076,Z 322.302,A -85,B 0,C 180,E1 -21803.321,E2 -21803.321} C_VEL
LIN {X 0,Y 215.512,Z 334.114,A -85,B 0,C 180,E1 -21805.084,E2 -21805.084} C_VEL
LIN {X 0,Y 211.895,Z 344.313,A -85,B 0,C 180,E1 -21807.056,E2 -21807.056} C_VEL
LIN {X 0,Y 208.031,Z 353.862,A -85,B 0,C 180,E1 -21809.436,E2 -21809.436} C_VEL
LIN {X 0,Y 204.662,Z 361.381,A -85,B 0,C 180,E1 -21811.798,E2 -21811.798} C_VEL
LIN {X 0,Y 200.928,Z 369.098,A -85,B 0,C 180,E1 -21814.876,E2 -21814.876} C_VEL
LIN {X 0,Y 197.392,Z 375.737,A -85,B 0,C 180,E1 -21818.436,E2 -21818.436} C_VEL
LIN {X 0,Y 194.535,Z 380.833,A -85,B 0,C 180,E1 -21822.216,E2 -21822.216} C_VEL
LIN {X 0,Y 192.41,Z 384.268,A -85,B 0,C 180,E1 -21826.052,E2 -21826.052} C_VEL
LIN {X 0,Y 191.354,Z 385.768,A -85,B 0,C 180,E1 -21828.616,E2 -21828.616} C_VEL
LIN {X 0,Y 190.599,Z 386.635,A -85,B 0,C 180,E1 -21831.182,E2 -21831.182} C_VEL
LIN {X 0,Y 189.969,Z 386.912,A -85,B 0,C 180,E1 -21834.479,E2 -21834.479} C_VEL
LIN {X 0,Y 189.75,Z 385.836,A -85,B 0,C 180,E1 -21838.766,E2 -21838.766} C_VEL
LIN {X 0,Y 190.095,Z 383.522,A -85,B 0,C 180,E1 -21842.537,E2 -21842.537} C_VEL
LIN {X 0,Y 190.837,Z 380.032,A -85,B 0,C 180,E1 -21846.102,E2 -21846.102} C_VEL
LIN {X 0,Y 191.77,Z 375.236,A -85,B 0,C 180,E1 -21849.625,E2 -21849.625} C_VEL
LIN {X 0,Y 193.204,Z 369.017,A -85,B 0,C 180,E1 -21853.081,E2 -21853.081} C_VEL
LIN {X 0,Y 194.87,Z 362.33,A -85,B 0,C 180,E1 -21855.99,E2 -21855.99} C_VEL
LIN {X 0,Y 196.813,Z 354.635,A -85,B 0,C 180,E1 -21858.673,E2 -21858.673} C_VEL
LIN {X 0,Y 199.24,Z 344.465,A -85,B 0,C 180,E1 -21861.492,E2 -21861.492} C_VEL
LIN {X 0,Y 201.616,Z 334.134,A -85,B 0,C 180,E1 -21863.746,E2 -21863.746} C_VEL
LIN {X 0,Y 203.939,Z 322.02,A -85,B 0,C 180,E1 -21865.8,E2 -21865.8} C_VEL
LIN {X 0,Y 205.976,Z 309.376,A -85,B 0,C 180,E1 -21867.433,E2 -21867.433} C_VEL
LIN {X 0,Y 207.671,Z 295.941,A -85,B 0,C 180,E1 -21868.667,E2 -21868.667} C_VEL
LIN {X 0,Y 208.902,Z 282.975,A -85,B 0,C 180,E1 -21869.458,E2 -21869.458} C_VEL
LIN {X 0,Y 211.811,Z 222.729,A -85,B 0,C 180,E1 -21871.603,E2 -21871.603} C_VEL
LIN {X 0,Y 202.764,Z 198.273,A -85,B 0,C 180,E1 -21874.005,E2 -21874.005} C_VEL
LIN {X 0,Y 193.868,Z 182.126,A -85,B 0,C 180,E1 -21876.244,E2 -21876.244} C_VEL
LIN {X 0,Y 192.957,Z 179.451,A -85,B 0,C 180,E1 -21876.536,E2 -21876.536} C_VEL
LIN {X 0,Y 192.938,Z 179.445,A -85,B 0,C 180,E1 -21880.494,E2 -21880.494} C_VEL
LIN {X 0,Y 192.728,Z 179.476,A -85,B 0,C 180,E1 -21884.789,E2 -21884.789} C_VEL
LIN {X 0,Y 192.663,Z 179.485,A -85,B 0,C 180,E1 -21889.166,E2 -21889.166} C_VEL
LIN {X 0,Y 192.612,Z 179.475,A -85,B 0,C 180,E1 -21894.189,E2 -21894.189} C_VEL
LIN {X 0,Y 192.602,Z 179.493,A -85,B 0,C 180,E1 -21898.865,E2 -21898.865} C_VEL
LIN {X 0,Y 192.596,Z 179.469,A -85,B 0,C 180,E1 -21903.187,E2 -21903.187} C_VEL
LIN {X 0,Y 192.545,Z 179.499,A -85,B 0,C 180,E1 -21908.354,E2 -21908.354} C_VEL
LIN {X 0,Y 192.486,Z 179.493,A -85,B 0,C 180,E1 -21913.094,E2 -21913.094} C_VEL
LIN {X 0,Y 192.485,Z 179.469,A -85,B 0,C 180,E1 -21916.907,E2 -21916.907} C_VEL
LIN {X 0,Y 192.543,Z 179.498,A -85,B 0,C 180,E1 -21921.646,E2 -21921.646} C_VEL
LIN {X 0,Y 192.596,Z 179.486,A -85,B 0,C 180,E1 -21926.813,E2 -21926.813} C_VEL
LIN {X 0,Y 192.623,Z 179.49,A -85,B 0,C 180,E1 -21931.685,E2 -21931.685} C_VEL
LIN {X 0,Y 192.673,Z 179.474,A -85,B 0,C 180,E1 -21936.344,E2 -21936.344} C_VEL
LIN {X 0,Y 192.696,Z 179.48,A -85,B 0,C 180,E1 -21941.492,E2 -21941.492} C_VEL
LIN {X 0,Y 192.781,Z 179.466,A -85,B 0,C 180,E1 -21947.365,E2 -21947.365} C_VEL
LIN {X 0,Y 193.029,Z 179.438,A -85,B 0,C 180,E1 -21951.626,E2 -21951.626} C_VEL
LIN {X 0,Y 193.233,Z 179.414,A -85,B 0,C 180,E1 -21957.916,E2 -21957.916} C_VEL
LIN {X 0,Y 193.416,Z 179.391,A -85,B 0,C 180,E1 -21960,E2 -21960} C_VEL
LIN {X 0,Y 192.937,Z 179.424,A -85,B 0,C 180,E1 -21964.178,E2 -21964.178} C_VEL
LIN {X 0,Y 193.024,Z 179.408,A -85,B 0,C 180,E1 -21968.374,E2 -21968.374} C_VEL
LIN {X 0,Y 192.773,Z 179.471,A -85,B 0,C 180,E1 -21972.635,E2 -21972.635} C_VEL
LIN {X 0,Y 192.696,Z 179.463,A -85,B 0,C 180,E1 -21978.508,E2 -21978.508} C_VEL
LIN {X 0,Y 192.627,Z 179.488,A -85,B 0,C 180,E1 -21984.198,E2 -21984.198} C_VEL
LIN {X 0,Y 192.602,Z 179.487,A -85,B 0,C 180,E1 -21988.865,E2 -21988.865} C_VEL
LIN {X 0,Y 192.596,Z 179.493,A -85,B 0,C 180,E1 -21993.186,E2 -21993.186} C_VEL
LIN {X 0,Y 192.543,Z 179.502,A -85,B 0,C 180,E1 -21998.354,E2 -21998.354} C_VEL
LIN {X 0,Y 192.486,Z 179.51,A -85,B 0,C 180,E1 -22003.093,E2 -22003.093} C_VEL
LIN {X 0,Y 192.577,Z 179.604,A -85,B 0,C 180,E1 -22008.531,E2 -22008.531} C_VEL
LIN {X 0,Y 193.984,Z 185.18,A -85,B 0,C 180,E1 -22011.517,E2 -22011.517} C_VEL
LIN {X 0,Y 202.638,Z 205.379,A -85,B 0,C 180,E1 -22013.88,E2 -22013.88} C_VEL
LIN {X 0,Y 208.831,Z 222.31,A -85,B 0,C 180,E1 -22015.55,E2 -22015.55} C_VEL
LIN {X 0,Y 211.126,Z 241.723,A -85,B 0,C 180,E1 -22016.684,E2 -22016.684} C_VEL
LIN {X 0,Y 210.631,Z 252.186,A -85,B 0,C 180,E1 -22017.05,E2 -22017.05} C_VEL
LIN {X 0,Y 209.795,Z 258.013,A -85,B 0,C 180,E1 -22017.18,E2 -22017.18} C_VEL
LIN {X 0,Y 203.725,Z 276.909,A -85,B 0,C 180,E1 -22017.151,E2 -22017.151} C_VEL
LIN {X 0,Y 202.831,Z 282.738,A -85,B 0,C 180,E1 -22017.278,E2 -22017.278} C_VEL
LIN {X 0,Y 201.818,Z 297.854,A -85,B 0,C 180,E1 -22017.931,E2 -22017.931} C_VEL
LIN {X 0,Y 200.396,Z 310.537,A -85,B 0,C 180,E1 -22018.849,E2 -22018.849} C_VEL
LIN {X 0,Y 198.625,Z 321.965,A -85,B 0,C 180,E1 -22020.014,E2 -22020.014} C_VEL
LIN {X 0,Y 196.654,Z 332.608,A -85,B 0,C 180,E1 -22021.445,E2 -22021.445} C_VEL
LIN {X 0,Y 194.167,Z 343.891,A -85,B 0,C 180,E1 -22023.389,E2 -22023.389} C_VEL
LIN {X 0,Y 191.832,Z 354.093,A -85,B 0,C 180,E1 -22025.659,E2 -22025.659} C_VEL
LIN {X 0,Y 189.423,Z 363.275,A -85,B 0,C 180,E1 -22028.221,E2 -22028.221} C_VEL
LIN {X 0,Y 187.996,Z 369.506,A -85,B 0,C 180,E1 -22030.339,E2 -22030.339} C_VEL
LIN {X 0,Y 186.032,Z 377.178,A -85,B 0,C 180,E1 -22033.54,E2 -22033.54} C_VEL
LIN {X 0,Y 184.582,Z 383.33,A -85,B 0,C 180,E1 -22036.794,E2 -22036.794} C_VEL
LIN {X 0,Y 183.713,Z 388.185,A -85,B 0,C 180,E1 -22040.087,E2 -22040.087} C_VEL
LIN {X 0,Y 183.228,Z 391.874,A -85,B 0,C 180,E1 -22043.392,E2 -22043.392} C_VEL
LIN {X 0,Y 183.08,Z 394.345,A -85,B 0,C 180,E1 -22046.451,E2 -22046.451} C_VEL
LIN {X 0,Y 183.202,Z 396.164,A -85,B 0,C 180,E1 -22050,E2 -22050} C_VEL
LIN {X 0,Y 183.053,Z 396.88,A -85,B 0,C 180,E1 -22053.414,E2 -22053.414} C_VEL
LIN {X 0,Y 183.212,Z 396.691,A -85,B 0,C 180,E1 -22056.608,E2 -22056.608} C_VEL
LIN {X 0,Y 184.06,Z 395.041,A -85,B 0,C 180,E1 -22061.006,E2 -22061.006} C_VEL
LIN {X 0,Y 184.806,Z 393.637,A -85,B 0,C 180,E1 -22063.19,E2 -22063.19} C_VEL
LIN {X 0,Y 186.39,Z 390.71,A -85,B 0,C 180,E1 -22066.427,E2 -22066.427} C_VEL
LIN {X 0,Y 188.673,Z 386.778,A -85,B 0,C 180,E1 -22069.588,E2 -22069.588} C_VEL
LIN {X 0,Y 191.442,Z 381.749,A -85,B 0,C 180,E1 -22072.673,E2 -22072.673} C_VEL
LIN {X 0,Y 194.638,Z 375.5,A -85,B 0,C 180,E1 -22075.677,E2 -22075.677} C_VEL
LIN {X 0,Y 198.497,Z 367.73,A -85,B 0,C 180,E1 -22078.554,E2 -22078.554} C_VEL
LIN {X 0,Y 202.966,Z 358.072,A -85,B 0,C 180,E1 -22081.292,E2 -22081.292} C_VEL
LIN {X 0,Y 206.966,Z 348.16,A -85,B 0,C 180,E1 -22083.491,E2 -22083.491} C_VEL
LIN {X 0,Y 210.967,Z 337.005,A -85,B 0,C 180,E1 -22085.368,E2 -22085.368} C_VEL
LIN {X 0,Y 214.207,Z 326.194,A -85,B 0,C 180,E1 -22086.782,E2 -22086.782} C_VEL
LIN {X 0,Y 217.074,Z 314.382,A -85,B 0,C 180,E1 -22087.963,E2 -22087.963} C_VEL
LIN {X 0,Y 219.573,Z 301.334,A -85,B 0,C 180,E1 -22088.864,E2 -22088.864} C_VEL
LIN {X 0,Y 221.11,Z 288.336,A -85,B 0,C 180,E1 -22089.473,E2 -22089.473} C_VEL
LIN {X 0,Y 224.06,Z 246.396,A -85,B 0,C 180,E1 -22090.889,E2 -22090.889} C_VEL
LIN {X 0,Y 223.538,Z 244.1,A -85,B 0,C 180,E1 -22091.171,E2 -22091.171} C_VEL
LIN {X 0,Y 219.874,Z 234.765,A -85,B 0,C 180,E1 -22092.845,E2 -22092.845} C_VEL
LIN {X 0,Y 215.29,Z 224.976,A -85,B 0,C 180,E1 -22095.047,E2 -22095.047} C_VEL
LIN {X 0,Y 210.828,Z 216.684,A -85,B 0,C 180,E1 -22097.353,E2 -22097.353} C_VEL
LIN {X 0,Y 207.285,Z 210.808,A -85,B 0,C 180,E1 -22099.384,E2 -22099.384} C_VEL
LIN {X 0,Y 204.167,Z 205.898,A -85,B 0,C 180,E1 -22101.323,E2 -22101.323} C_VEL
LIN {X 0,Y 200.923,Z 200.9,A -85,B 0,C 180,E1 -22103.62,E2 -22103.62} C_VEL
LIN {X 0,Y 197.173,Z 195.502,A -85,B 0,C 180,E1 -22106.698,E2 -22106.698} C_VEL
LIN {X 0,Y 196.138,Z 194.257,A -85,B 0,C 180,E1 -22107.64,E2 -22107.64} C_VEL
LIN {X 0,Y 191.552,Z 188.036,A -85,B 0,C 180,E1 -22112.997,E2 -22112.997} C_VEL
LIN {X 0,Y 189.469,Z 185.827,A -85,B 0,C 180,E1 -22116.5,E2 -22116.5} C_VEL
LIN {X 0,Y 187.683,Z 184.523,A -85,B 0,C 180,E1 -22122.568,E2 -22122.568} C_VEL
LIN {X 0,Y 187.859,Z 184.602,A -85,B 0,C 180,E1 -22127.029,E2 -22127.029} C_VEL
LIN {X 0,Y 190.774,Z 186.164,A -85,B 0,C 180,E1 -22134.084,E2 -22134.084} C_VEL
LIN {X 0,Y 191.5,Z 186.604,A -85,B 0,C 180,E1 -22135.138,E2 -22135.138} C_VEL
LIN {X 0,Y 192.829,Z 189.181,A -85,B 0,C 180,E1 -22137.128,E2 -22137.128} C_VEL
LIN {X 0,Y 195.97,Z 191.835,A -85,B 0,C 180,E1 -22140.395,E2 -22140.395} C_VEL
LIN {X 0,Y 196.427,Z 192.544,A -85,B 0,C 180,E1 -22140.847,E2 -22140.847} C_VEL
LIN {X 0,Y 198.212,Z 195.637,A -85,B 0,C 180,E1 -22142.54,E2 -22142.54} C_VEL
LIN {X 0,Y 200.562,Z 197.898,A -85,B 0,C 180,E1 -22144.333,E2 -22144.333} C_VEL
LIN {X 0,Y 203.218,Z 201.558,A -85,B 0,C 180,E1 -22146.242,E2 -22146.242} C_VEL
LIN {X 0,Y 204.373,Z 202.99,A -85,B 0,C 180,E1 -22147.005,E2 -22147.005} C_VEL
LIN {X 0,Y 208.004,Z 208.235,A -85,B 0,C 180,E1 -22149.22,E2 -22149.22} C_VEL
LIN {X 0,Y 210.943,Z 212.517,A -85,B 0,C 180,E1 -22150.859,E2 -22150.859} C_VEL
LIN {X 0,Y 214.91,Z 219.126,A -85,B 0,C 180,E1 -22152.892,E2 -22152.892} C_VEL
LIN {X 0,Y 220.134,Z 229.131,A -85,B 0,C 180,E1 -22155.375,E2 -22155.375} C_VEL
LIN {X 0,Y 224.177,Z 238.197,A -85,B 0,C 180,E1 -22157.158,E2 -22157.158} C_VEL
LIN {X 0,Y 224.602,Z 239.223,A -85,B 0,C 180,E1 -22157.342,E2 -22157.342} C_VEL
LIN {X 0,Y 221.112,Z 285.009,A -85,B 0,C 180,E1 -22158.869,E2 -22158.869} C_VEL
LIN {X 0,Y 219.204,Z 298.615,A -85,B 0,C 180,E1 -22159.641,E2 -22159.641} C_VEL
LIN {X 0,Y 217.049,Z 309.894,A -85,B 0,C 180,E1 -22160.596,E2 -22160.596} C_VEL
LIN {X 0,Y 214.025,Z 322.069,A -85,B 0,C 180,E1 -22161.982,E2 -22161.982} C_VEL
LIN {X 0,Y 210.594,Z 333.056,A -85,B 0,C 180,E1 -22163.608,E2 -22163.608} C_VEL
LIN {X 0,Y 206.794,Z 343.472,A -85,B 0,C 180,E1 -22165.593,E2 -22165.593} C_VEL
LIN {X 0,Y 202.796,Z 352.943,A -85,B 0,C 180,E1 -22167.905,E2 -22167.905} C_VEL
LIN {X 0,Y 198.475,Z 362.121,A -85,B 0,C 180,E1 -22170.829,E2 -22170.829} C_VEL
LIN {X 0,Y 194.688,Z 369.463,A -85,B 0,C 180,E1 -22173.873,E2 -22173.873} C_VEL
LIN {X 0,Y 191.412,Z 375.232,A -85,B 0,C 180,E1 -22177.004,E2 -22177.004} C_VEL
LIN {X 0,Y 188.65,Z 379.807,A -85,B 0,C 180,E1 -22180.291,E2 -22180.291} C_VEL
LIN {X 0,Y 186.203,Z 383.631,A -85,B 0,C 180,E1 -22184.181,E2 -22184.181} C_VEL
LIN {X 0,Y 184.915,Z 385.402,A -85,B 0,C 180,E1 -22186.833,E2 -22186.833} C_VEL
LIN {X 0,Y 183.832,Z 386.665,A -85,B 0,C 180,E1 -22189.873,E2 -22189.873} C_VEL
LIN {X 0,Y 182.952,Z 387.14,A -85,B 0,C 180,E1 -22193.776,E2 -22193.776} C_VEL
LIN {X 0,Y 182.645,Z 386.3,A -85,B 0,C 180,E1 -22197.838,E2 -22197.838} C_VEL
LIN {X 0,Y 182.919,Z 383.981,A -85,B 0,C 180,E1 -22202.092,E2 -22202.092} C_VEL
LIN {X 0,Y 183.473,Z 381.371,A -85,B 0,C 180,E1 -22205.079,E2 -22205.079} C_VEL
LIN {X 0,Y 184.396,Z 376.969,A -85,B 0,C 180,E1 -22208.772,E2 -22208.772} C_VEL
LIN {X 0,Y 185.671,Z 371.185,A -85,B 0,C 180,E1 -22212.373,E2 -22212.373} C_VEL
LIN {X 0,Y 187.441,Z 364.251,A -85,B 0,C 180,E1 -22215.693,E2 -22215.693} C_VEL
LIN {X 0,Y 189.646,Z 356.069,A -85,B 0,C 180,E1 -22218.781,E2 -22218.781} C_VEL
LIN {X 0,Y 191.955,Z 346.715,A -85,B 0,C 180,E1 -22221.579,E2 -22221.579} C_VEL
LIN {X 0,Y 194.476,Z 336.229,A -85,B 0,C 180,E1 -22224.036,E2 -22224.036} C_VEL
LIN {X 0,Y 196.781,Z 325.253,A -85,B 0,C 180,E1 -22226.071,E2 -22226.071} C_VEL
LIN {X 0,Y 198.887,Z 313.49,A -85,B 0,C 180,E1 -22227.748,E2 -22227.748} C_VEL
LIN {X 0,Y 200.678,Z 300.598,A -85,B 0,C 180,E1 -22229.122,E2 -22229.122} C_VEL
LIN {X 0,Y 202.116,Z 287.777,A -85,B 0,C 180,E1 -22230.058,E2 -22230.058} C_VEL
LIN {X 0,Y 203.114,Z 271.868,A -85,B 0,C 180,E1 -22230.749,E2 -22230.749} C_VEL
LIN {X 0,Y 205.424,Z 224.136,A -85,B 0,C 180,E1 -22232.468,E2 -22232.468} C_VEL
LIN {X 0,Y 197.148,Z 201.683,A -85,B 0,C 180,E1 -22234.765,E2 -22234.765} C_VEL
LIN {X 0,Y 186.136,Z 181.219,A -85,B 0,C 180,E1 -22237.729,E2 -22237.729} C_VEL
LIN {X 0,Y 185.981,Z 180.319,A -85,B 0,C 180,E1 -22237.873,E2 -22237.873} C_VEL
LIN {X 0,Y 185.847,Z 180.326,A -85,B 0,C 180,E1 -22240.899,E2 -22240.899} C_VEL
LIN {X 0,Y 185.66,Z 180.351,A -85,B 0,C 180,E1 -22245.366,E2 -22245.366} C_VEL
LIN {X 0,Y 185.559,Z 180.373,A -85,B 0,C 180,E1 -22249.93,E2 -22249.93} C_VEL
LIN {X 0,Y 185.546,Z 180.355,A -85,B 0,C 180,E1 -22254.624,E2 -22254.624} C_VEL
LIN {X 0,Y 185.545,Z 180.371,A -85,B 0,C 180,E1 -22259.499,E2 -22259.499} C_VEL
LIN {X 0,Y 185.499,Z 180.354,A -85,B 0,C 180,E1 -22264.632,E2 -22264.632} C_VEL
LIN {X 0,Y 185.503,Z 180.372,A -85,B 0,C 180,E1 -22267.314,E2 -22267.314} C_VEL
LIN {X 0,Y 185.464,Z 180.382,A -85,B 0,C 180,E1 -22270.722,E2 -22270.722} C_VEL
LIN {X 0,Y 185.456,Z 180.342,A -85,B 0,C 180,E1 -22276.057,E2 -22276.057} C_VEL
LIN {X 0,Y 185.457,Z 180.368,A -85,B 0,C 180,E1 -22279.892,E2 -22279.892} C_VEL
LIN {X 0,Y 185.502,Z 180.376,A -85,B 0,C 180,E1 -22282.714,E2 -22282.714} C_VEL
LIN {X 0,Y 185.533,Z 180.361,A -85,B 0,C 180,E1 -22287.973,E2 -22287.973} C_VEL
LIN {X 0,Y 185.549,Z 180.369,A -85,B 0,C 180,E1 -22290.595,E2 -22290.595} C_VEL
LIN {X 0,Y 185.582,Z 180.359,A -85,B 0,C 180,E1 -22295.382,E2 -22295.382} C_VEL
LIN {X 0,Y 185.627,Z 180.362,A -85,B 0,C 180,E1 -22301.179,E2 -22301.179} C_VEL
LIN {X 0,Y 185.704,Z 180.345,A -85,B 0,C 180,E1 -22306.875,E2 -22306.875} C_VEL
LIN {X 0,Y 185.978,Z 180.316,A -85,B 0,C 180,E1 -22311.306,E2 -22311.306} C_VEL
LIN {X 0,Y 186.179,Z 180.293,A -85,B 0,C 180,E1 -22317.837,E2 -22317.837} C_VEL
LIN {X 0,Y 186.382,Z 180.267,A -85,B 0,C 180,E1 -22320,E2 -22320} C_VEL
LIN {X 0,Y 185.885,Z 180.3,A -85,B 0,C 180,E1 -22324.337,E2 -22324.337} C_VEL
LIN {X 0,Y 185.974,Z 180.288,A -85,B 0,C 180,E1 -22328.694,E2 -22328.694} C_VEL
LIN {X 0,Y 185.698,Z 180.352,A -85,B 0,C 180,E1 -22333.125,E2 -22333.125} C_VEL
LIN {X 0,Y 185.627,Z 180.338,A -85,B 0,C 180,E1 -22338.821,E2 -22338.821} C_VEL
LIN {X 0,Y 185.562,Z 180.368,A -85,B 0,C 180,E1 -22344.635,E2 -22344.635} C_VEL
LIN {X 0,Y 185.545,Z 180.368,A -85,B 0,C 180,E1 -22349.499,E2 -22349.499} C_VEL
LIN {X 0,Y 185.498,Z 180.377,A -85,B 0,C 180,E1 -22354.632,E2 -22354.632} C_VEL
LIN {X 0,Y 185.5,Z 180.38,A -85,B 0,C 180,E1 -22357.314,E2 -22357.314} C_VEL
LIN {X 0,Y 185.462,Z 180.382,A -85,B 0,C 180,E1 -22360.721,E2 -22360.721} C_VEL
LIN {X 0,Y 185.456,Z 180.373,A -85,B 0,C 180,E1 -22366.056,E2 -22366.056} C_VEL
LIN {X 0,Y 185.498,Z 180.468,A -85,B 0,C 180,E1 -22367.628,E2 -22367.628} C_VEL
LIN {X 0,Y 186.596,Z 184.894,A -85,B 0,C 180,E1 -22370.143,E2 -22370.143} C_VEL
LIN {X 0,Y 194.388,Z 202.36,A -85,B 0,C 180,E1 -22372.392,E2 -22372.392} C_VEL
LIN {X 0,Y 201.54,Z 220.931,A -85,B 0,C 180,E1 -22374.395,E2 -22374.395} C_VEL
LIN {X 0,Y 202.888,Z 225.717,A -85,B 0,C 180,E1 -22374.814,E2 -22374.814} C_VEL
LIN {X 0,Y 204.786,Z 242.037,A -85,B 0,C 180,E1 -22375.806,E2 -22375.806} C_VEL
LIN {X 0,Y 202.831,Z 282.738,A -85,B 0,C 180,E1 -22377.278,E2 -22377.278} C_VEL
LIN {X 0,Y 201.878,Z 288.552,A -85,B 0,C 180,E1 -22377.403,E2 -22377.403} C_VEL
LIN {X 0,Y 198.525,Z 297.893,A -85,B 0,C 180,E1 -22377.487,E2 -22377.487} C_VEL
LIN {X 0,Y 194.934,Z 307.095,A -85,B 0,C 180,E1 -22377.783,E2 -22377.783} C_VEL
LIN {X 0,Y 193.602,Z 312.687,A -85,B 0,C 180,E1 -22378.205,E2 -22378.205} C_VEL
LIN {X 0,Y 191.723,Z 323.786,A -85,B 0,C 180,E1 -22379.428,E2 -22379.428} C_VEL
LIN {X 0,Y 189.709,Z 334.027,A -85,B 0,C 180,E1 -22380.907,E2 -22380.907} C_VEL
LIN {X 0,Y 187.221,Z 344.972,A -85,B 0,C 180,E1 -22382.925,E2 -22382.925} C_VEL
LIN {X 0,Y 184.563,Z 356,A -85,B 0,C 180,E1 -22385.566,E2 -22385.566} C_VEL
LIN {X 0,Y 182.281,Z 364.541,A -85,B 0,C 180,E1 -22388.137,E2 -22388.137} C_VEL
LIN {X 0,Y 180.147,Z 372.739,A -85,B 0,C 180,E1 -22391.225,E2 -22391.225} C_VEL
LIN {X 0,Y 178.298,Z 379.725,A -85,B 0,C 180,E1 -22394.57,E2 -22394.57} C_VEL
LIN {X 0,Y 176.944,Z 386.13,A -85,B 0,C 180,E1 -22398.545,E2 -22398.545} C_VEL
LIN {X 0,Y 176.313,Z 390.289,A -85,B 0,C 180,E1 -22401.98,E2 -22401.98} C_VEL
LIN {X 0,Y 175.996,Z 394.201,A -85,B 0,C 180,E1 -22406.681,E2 -22406.681} C_VEL
